(* IEC 61131-3 sources: OpenPLC_Sample_Programs/successed_ST (part 13) *)

(* ---- Scenario3v1_Final.st ---- *)
TYPE
    STATES_CRANE : (INIT, START_CRANE, CRANE_INIT, CRANE_INIT_2, INTERSTEP, INTERSTEP_2, TIMEDELAY, TURN_RIGHT, INTERSTEP_CHECK_WORKPIECE, CRANE_LOWER, STEP0, CRANE_LIFT_MAGAZIN, CRANE_TURN_LEFT_NOT_METALLIC, CRANE_ON_CONVEYOR, CRANE_LIFT_MAGAZIN_METALLIC, CRANE_TURN_LEFT_METALLIC, CRANE_ON_STAMP_METALLIC, RELEASE_WORKPIECE, CRANE_GO_UP, PAUSE, RESET_INTERCONNECT, LOWER_CRANE, SUCK_AT_STAMP, CRANE_LIFT_AT_STAMP, CRANE_TURN_LEFT_FROM_STAMP, CRANE_ON_CONVEYOR_METALLIC, RELEASE, CRANE_LIFT_CONVEYOR, WAIT_AT_STAMP, STEP2);
    STATES_MAGAZIN : (INIT, START_MAGAZIN, GREEN_LAMP, MAGAZIN_INIT, MAGAZIN_INIT_2, INTERSTEP, CONVEY, STEP0, SLIDER_MOVE_BACK, STEP1);
    STATES_STAMP : (INIT, START_STAMP, GREEN_LAMP, STAMP_INIT_1, STAMP_INIT_2, STAMP_INIT_3, STAMP_INIT_4, INTERSTEP, INTERSTEP_2, STEP0, STAMPSLIDERBACK, STAMPPROCESS, STEP1, STAMPSLIDERFORWARD, STEP2);
END_TYPE

PROGRAM MAIN
    VAR_OUTPUT
        ACTUATOR_ANALOGCRANEPRESSURE : INT := INT#0;
        ACTUATOR_CRANELOWER : BOOL := FALSE;
        ACTUATOR_CRANETURNCLOCKWISE : BOOL := FALSE;
        ACTUATOR_CRANETURNCOUNTERCLOCKWISE : BOOL := FALSE;
        ACTUATOR_MAGAZINGREENLAMP : BOOL := FALSE;
        ACTUATOR_MAGAZINSLIDER : BOOL := FALSE;
        ACTUATOR_MAGAZINVACUUMOFF : BOOL := FALSE;
        ACTUATOR_MAGAZINVACUUMON : BOOL := FALSE;
        ACTUATOR_MAGAZINWHITELAMP : BOOL := FALSE;
        ACTUATOR_SOMEACTUATOR : BOOL := FALSE;
        ACTUATOR_STAMPGREENLAMP : BOOL := FALSE;
        ACTUATOR_STAMPPUSHER : BOOL := FALSE;
        ACTUATOR_STAMPSLIDERMOVEDIN : BOOL := FALSE;
        ACTUATOR_STAMPSLIDERMOVEDOUT : BOOL := FALSE;
        ACTUATOR_STAMPWHITELAMP : BOOL := FALSE;
    END_VAR

    VAR
        CRANE_CRANEDOWN : BOOL := FALSE;
        CRANE_CRANELOWER : BOOL := FALSE;
        CRANE_CRANEONCONVEYOR : BOOL := FALSE;
        CRANE_CRANEONMAGAZIN : BOOL := FALSE;
        CRANE_CRANEPOSITIONSTAMP : BOOL := FALSE;
        CRANE_CRANESUCKED : BOOL := FALSE;
        CRANE_CRANETURNCLOCKWISE : BOOL := FALSE;
        CRANE_CRANETURNCOUNTERCLOCKWISE : BOOL := FALSE;
        CRANE_CRANEUP : BOOL := FALSE;
        CRANE_DURATION1 : UINT := UINT#0;
        CRANE_MAGAZINCAPACITIVESENSOR : BOOL := FALSE;
        CRANE_MAGAZINVACUUMOFF : BOOL := FALSE;
        CRANE_MAGAZINVACUUMON : BOOL := FALSE;
        CRANE_SFCINIT : BOOL := FALSE;
        CRANE_SFCRESET : BOOL := FALSE;
        CRANE_SLIDERMOVEDOUT : BOOL := FALSE;
        CRANE_SLIDERNOTMOVEDOUT : BOOL := FALSE;
        CRANE_STAMPLOWERED : BOOL := FALSE;
        CRANE_STAMPSLIDERFILLED : BOOL := FALSE;
        CRANE_STARTBUTTONMAGAZIN : BOOL := FALSE;
        CRANE_STARTCOMMANDCRANE : BOOL := FALSE;
        CRANE_STARTVAR : BOOL := FALSE;
        CRANE_TIMEDELAY_TIMER_ET : UINT := UINT#0;
        CRANE_TIMEDELAY_TIMER_IN : BOOL := FALSE;
        CRANE_TIMEDELAY_TIMER_PT : UINT := UINT#0;
        CRANE_TIMEDELAY_TIMER_Q : BOOL := FALSE;
        CRANE_TIMEDELAY_TIMER_DURATION : UINT := UINT#0;
        CRANE_TIMEDELAY_TIMER_INTERCONNECT : BOOL := FALSE;
        CRANE_TIMER1_ET : UINT := UINT#0;
        CRANE_TIMER1_IN : BOOL := FALSE;
        CRANE_TIMER1_PT : UINT := UINT#0;
        CRANE_TIMER1_Q : BOOL := FALSE;
        CRANE_WORKPIECEREADY : BOOL := FALSE;
        CRANE_2_TRANSIT : BOOL := FALSE;
        CRANE_2STATE : STATES_CRANE := STATES_CRANE#INIT;
        CRANE_ACTUALTIME1 : UINT := UINT#0;
        CRANE_INTERCONNECT : BOOL := FALSE;
        CRANE_INTERCONNECTCRANESTARTCOMMAND : BOOL := FALSE;
        MAG_CRANEDOWN : BOOL := FALSE;
        MAG_CRANELOWER : BOOL := FALSE;
        MAG_CRANEONCONVEYOR : BOOL := FALSE;
        MAG_CRANEONMAGAZIN : BOOL := FALSE;
        MAG_CRANESUCKED : BOOL := FALSE;
        MAG_CRANETURNCLOCKWISE : BOOL := FALSE;
        MAG_CRANETURNCOUNTERCLOCKWISE : BOOL := FALSE;
        MAG_CRANEUP : BOOL := FALSE;
        MAG_MAGAZINGREENLAMP : BOOL := FALSE;
        MAG_MAGAZINSLIDER : BOOL := FALSE;
        MAG_MAGAZINVACUUMOFF : BOOL := FALSE;
        MAG_MAGAZINVACUUMON : BOOL := FALSE;
        MAG_MAGAZINWHITELAMP : BOOL := FALSE;
        MAG_SFCINIT : BOOL := FALSE;
        MAG_SFCRESET : BOOL := FALSE;
        MAG_SLIDERMOVEDOUT : BOOL := FALSE;
        MAG_SLIDERNOTMOVEDOUT : BOOL := FALSE;
        MAG_STARTBUTTONMAGAZIN : BOOL := FALSE;
        MAG_STARTCOMMANDMAGAZIN : BOOL := FALSE;
        MAG_STARTVAR : BOOL := FALSE;
        MAG_WORKPIECEREADY : BOOL := FALSE;
        MAG_2_TRANSIT : BOOL := FALSE;
        MAG_2STATE : STATES_MAGAZIN := STATES_MAGAZIN#INIT;
        MAG_INTERCONNECTMAGAZINSTARTCOMMAND : BOOL := FALSE;
        STAMP_CRANEDOWN : BOOL := FALSE;
        STAMP_CRANEONCONVEYOR : BOOL := FALSE;
        STAMP_CRANEPOSITIONSTAMP : BOOL := FALSE;
        STAMP_CRANESUCKED : BOOL := FALSE;
        STAMP_CRANEUP : BOOL := FALSE;
        STAMP_DURATION : UINT := UINT#0;
        STAMP_SFCINIT : BOOL := FALSE;
        STAMP_SFCRESET : BOOL := FALSE;
        STAMP_STAMPGREENLAMP : BOOL := FALSE;
        STAMP_STAMPLOWERED : BOOL := FALSE;
        STAMP_STAMPPRESSURE : BOOL := FALSE;
        STAMP_STAMPPUSHER : BOOL := FALSE;
        STAMP_STAMPSLIDERFILLED : BOOL := FALSE;
        STAMP_STAMPSLIDERMOVEDIN : BOOL := FALSE;
        STAMP_STAMPSLIDERMOVEDOUT : BOOL := FALSE;
        STAMP_STAMPSLIDERSENSORMOVEDIN : BOOL := FALSE;
        STAMP_STAMPSLIDERSENSORMOVEDOUT : BOOL := FALSE;
        STAMP_STAMPSTARTBUTTON : BOOL := FALSE;
        STAMP_STAMPUP : BOOL := FALSE;
        STAMP_STAMPWHITELAMP : BOOL := FALSE;
        STAMP_STARTCOMMANDSTAMP : BOOL := FALSE;
        STAMP_STARTVAR : BOOL := FALSE;
        STAMP_TIMER_ET : UINT := UINT#0;
        STAMP_TIMER_IN : BOOL := FALSE;
        STAMP_TIMER_PT : UINT := UINT#0;
        STAMP_TIMER_Q : BOOL := FALSE;
        STAMP_2_TRANSIT : BOOL := FALSE;
        STAMP_2STATE : STATES_STAMP := STATES_STAMP#INIT;
        STAMP_INTERCONNECT : BOOL := FALSE;
        STAMP_INTERCONNECTSTAMPSTARTCOMMAND : BOOL := FALSE;
    END_VAR

    VAR
        CRANE_SFCPAUSE : BOOL := FALSE;
        MAG_SFCPAUSE : BOOL := FALSE;
        STAMP_SFCPAUSE : BOOL := FALSE;
    END_VAR

    VAR_INPUT
        SENSOR_CRANEDOWN : BOOL := FALSE;
        SENSOR_CRANEONCONVEYOR : BOOL := FALSE;
        SENSOR_CRANEONMAGAZIN : BOOL := FALSE;
        SENSOR_CRANEPOSITION : BOOL := FALSE;
        SENSOR_CRANEPOSITIONSTAMP : BOOL := FALSE;
        SENSOR_CRANESUCKED : BOOL := FALSE;
        SENSOR_CRANEUP : BOOL := FALSE;
        SENSOR_MAGAZINCAPACITIVESENSOR : BOOL := FALSE;
        SENSOR_MAGAZINEMERGENCYSTOP : BOOL := FALSE;
        SENSOR_MAGAZINOPTICALSENSOR : BOOL := FALSE;
        SENSOR_MAGAZINSWITCHMANUELLAUTOMATIC : BOOL := FALSE;
        SENSOR_SLIDERMOVEDOUT : BOOL := FALSE;
        SENSOR_SLIDERNOTMOVEDOUT : BOOL := FALSE;
        SENSOR_STAMPEMERGENCYSTOP : BOOL := FALSE;
        SENSOR_STAMPLOWERED : BOOL := FALSE;
        SENSOR_STAMPSLIDERFILLED : BOOL := FALSE;
        SENSOR_STAMPSLIDERSENSORMOVEDIN : BOOL := FALSE;
        SENSOR_STAMPSLIDERSENSORMOVEDOUT : BOOL := FALSE;
        SENSOR_STAMPSTARTBUTTON : BOOL := FALSE;
        SENSOR_STAMPSWITCHMANUELLAUTOMATIC : BOOL := FALSE;
        SENSOR_STAMPUP : BOOL := FALSE;
        SENSOR_STARTBUTTONMAGAZIN : BOOL := FALSE;
        SENSOR_WORKPIECEREADY : BOOL := FALSE;
    END_VAR

    MAG_SLIDERNOTMOVEDOUT := SENSOR_SLIDERNOTMOVEDOUT;
    MAG_SLIDERMOVEDOUT := SENSOR_SLIDERMOVEDOUT;
    MAG_CRANEONMAGAZIN := SENSOR_CRANEONMAGAZIN;
    MAG_CRANEDOWN := SENSOR_CRANEDOWN;
    MAG_CRANEUP := SENSOR_CRANEUP;
    MAG_CRANEONCONVEYOR := SENSOR_CRANEONCONVEYOR;
    MAG_WORKPIECEREADY := SENSOR_WORKPIECEREADY;
    MAG_STARTBUTTONMAGAZIN := SENSOR_STARTBUTTONMAGAZIN;
    ACTUATOR_MAGAZINSLIDER := MAG_MAGAZINSLIDER;
    ACTUATOR_MAGAZINGREENLAMP := MAG_MAGAZINGREENLAMP;
    CRANE_CRANEUP := SENSOR_CRANEUP;
    CRANE_CRANEONCONVEYOR := SENSOR_CRANEONCONVEYOR;
    CRANE_CRANEDOWN := SENSOR_CRANEDOWN;
    CRANE_CRANESUCKED := SENSOR_CRANESUCKED;
    CRANE_CRANEONMAGAZIN := SENSOR_CRANEONMAGAZIN;
    CRANE_MAGAZINCAPACITIVESENSOR := SENSOR_MAGAZINCAPACITIVESENSOR;
    CRANE_CRANEPOSITIONSTAMP := SENSOR_CRANEPOSITIONSTAMP;
    CRANE_SLIDERMOVEDOUT := SENSOR_SLIDERMOVEDOUT;
    CRANE_WORKPIECEREADY := SENSOR_WORKPIECEREADY;
    CRANE_STAMPSLIDERFILLED := SENSOR_STAMPSLIDERFILLED;
    CRANE_SLIDERMOVEDOUT := SENSOR_SLIDERMOVEDOUT;
    CRANE_STARTBUTTONMAGAZIN := SENSOR_STARTBUTTONMAGAZIN;
    ACTUATOR_CRANETURNCOUNTERCLOCKWISE := CRANE_CRANETURNCOUNTERCLOCKWISE;
    ACTUATOR_CRANETURNCLOCKWISE := CRANE_CRANETURNCLOCKWISE;
    ACTUATOR_CRANELOWER := CRANE_CRANELOWER;
    ACTUATOR_MAGAZINVACUUMOFF := CRANE_MAGAZINVACUUMOFF;
    ACTUATOR_MAGAZINVACUUMON := CRANE_MAGAZINVACUUMON;
    STAMP_STAMPSLIDERSENSORMOVEDOUT := SENSOR_STAMPSLIDERSENSORMOVEDOUT;
    STAMP_STAMPSLIDERSENSORMOVEDIN := SENSOR_STAMPSLIDERSENSORMOVEDIN;
    STAMP_STAMPSLIDERFILLED := SENSOR_STAMPSLIDERFILLED;
    STAMP_STAMPUP := SENSOR_STAMPUP;
    STAMP_STAMPLOWERED := SENSOR_STAMPLOWERED;
    STAMP_CRANEDOWN := SENSOR_CRANEDOWN;
    STAMP_CRANEUP := SENSOR_CRANEUP;
    STAMP_CRANESUCKED := SENSOR_CRANESUCKED;
    STAMP_CRANEPOSITIONSTAMP := SENSOR_CRANEPOSITIONSTAMP;
    STAMP_CRANEONCONVEYOR := SENSOR_CRANEONCONVEYOR;
    STAMP_STAMPSTARTBUTTON := SENSOR_STAMPSTARTBUTTON;
    ACTUATOR_STAMPSLIDERMOVEDOUT := STAMP_STAMPSLIDERMOVEDOUT;
    ACTUATOR_STAMPSLIDERMOVEDIN := STAMP_STAMPSLIDERMOVEDIN;
    ACTUATOR_STAMPWHITELAMP := STAMP_STAMPWHITELAMP;
    ACTUATOR_STAMPPUSHER := STAMP_STAMPPUSHER;
    ACTUATOR_STAMPGREENLAMP := STAMP_STAMPGREENLAMP;
    ACTUATOR_ANALOGCRANEPRESSURE := INT#6000;
    IF (SENSOR_STAMPEMERGENCYSTOP AND SENSOR_MAGAZINEMERGENCYSTOP) THEN
        (* ! REGION MAG[MAG_SFCINIT, MAG_INTERCONNECTMAGAZINSTARTCOMMAND](MAG_CRANEDOWN, MAG_CRANEONCONVEYOR, MAG_CRANEONMAGAZIN, MAG_CRANESUCKED, MAG_CRANEUP, MAG_SFCRESET, MAG_SLIDERMOVEDOUT, MAG_SLIDERNOTMOVEDOUT, MAG_STARTBUTTONMAGAZIN, MAG_STARTVAR, MAG_WORKPIECEREADY) => (MAG_CRANELOWER, MAG_CRANETURNCLOCKWISE, MAG_CRANETURNCOUNTERCLOCKWISE, MAG_MAGAZINGREENLAMP, MAG_MAGAZINSLIDER, MAG_MAGAZINVACUUMOFF, MAG_MAGAZINVACUUMON, MAG_MAGAZINWHITELAMP, MAG_STARTCOMMANDMAGAZIN)
 *)            IF (MAG_SFCINIT OR MAG_SFCRESET) THEN
                MAG_CRANEDOWN := FALSE;
                MAG_CRANELOWER := FALSE;
                MAG_CRANEONCONVEYOR := FALSE;
                MAG_CRANEONMAGAZIN := FALSE;
                MAG_CRANESUCKED := FALSE;
                MAG_CRANETURNCLOCKWISE := FALSE;
                MAG_CRANETURNCOUNTERCLOCKWISE := FALSE;
                MAG_CRANEUP := FALSE;
                MAG_MAGAZINGREENLAMP := FALSE;
                MAG_MAGAZINSLIDER := FALSE;
                MAG_MAGAZINVACUUMOFF := FALSE;
                MAG_MAGAZINVACUUMON := FALSE;
                MAG_MAGAZINWHITELAMP := FALSE;
                MAG_SFCINIT := FALSE;
                MAG_SFCRESET := FALSE;
                MAG_SLIDERMOVEDOUT := FALSE;
                MAG_SLIDERNOTMOVEDOUT := FALSE;
                MAG_STARTBUTTONMAGAZIN := FALSE;
                MAG_STARTCOMMANDMAGAZIN := FALSE;
                MAG_STARTVAR := FALSE;
                MAG_WORKPIECEREADY := FALSE;
                MAG_2_TRANSIT := FALSE;
                MAG_2STATE := STATES_MAGAZIN#INIT;
                MAG_INTERCONNECTMAGAZINSTARTCOMMAND := FALSE;
            END_IF;
            IF NOT (MAG_SFCINIT OR MAG_SFCPAUSE) THEN
                (* RUNNING PIPELINE STEP: EDU.KIT.ITI.FORMAL.AUTOMATION.ST.INTRODUCESTATEENUMVARIABLE
 *)
                (* END OF: EDU.KIT.ITI.FORMAL.AUTOMATION.ST.INTRODUCESTATEENUMVARIABLE
 *)
                (* RUNNING PIPELINE STEP: EDU.KIT.ITI.FORMAL.AUTOMATION.ST.TRANSLATIONSFCTOSTOLD_INTRODUCETRANSITVARIABLE
 *)
                (* END OF: EDU.KIT.ITI.FORMAL.AUTOMATION.ST.TRANSLATIONSFCTOSTOLD_INTRODUCETRANSITVARIABLE
 *)
                (* RUNNING PIPELINE STEP: EDU.KIT.ITI.FORMAL.AUTOMATION.ST.TRANSLATIONSFCTOSTOLD_THEBIGSTATECASE
 *)
                CASE MAG_2STATE OF
                    STATES_MAGAZIN#INIT:
                        MAG_2_TRANSIT := FALSE;
                        IF TRUE THEN
                            MAG_2_TRANSIT := TRUE;
                            MAG_2STATE := STATES_MAGAZIN#START_MAGAZIN;
                        END_IF;

                    STATES_MAGAZIN#START_MAGAZIN:
                        MAG_2_TRANSIT := FALSE;
                        (* CALL OF ACTION: START_MAGAZIN_ACTIVE
 *)
                        MAG_MAGAZINSLIDER := FALSE;
                        MAG_MAGAZINGREENLAMP := FALSE;
                        MAG_STARTVAR := FALSE;
                        MAG_STARTCOMMANDMAGAZIN := FALSE;
                        IF (MAG_STARTBUTTONMAGAZIN = TRUE) THEN
                            MAG_INTERCONNECTMAGAZINSTARTCOMMAND := TRUE;
                        END_IF;
                        (* END OF ACTION CALL: START_MAGAZIN_ACTIVE
 *)
                        IF MAG_INTERCONNECTMAGAZINSTARTCOMMAND THEN
                            MAG_2_TRANSIT := TRUE;
                            MAG_2STATE := STATES_MAGAZIN#GREEN_LAMP;
                        END_IF;

                    STATES_MAGAZIN#GREEN_LAMP:
                        MAG_2_TRANSIT := FALSE;
                        (* CALL OF ACTION: GREEN_LAMP_ACTIVE
 *)
                        MAG_MAGAZINGREENLAMP := TRUE;
                        MAG_INTERCONNECTMAGAZINSTARTCOMMAND := FALSE;
                        (* END OF ACTION CALL: GREEN_LAMP_ACTIVE
 *)
                        IF TRUE THEN
                            MAG_2_TRANSIT := TRUE;
                            MAG_2STATE := STATES_MAGAZIN#MAGAZIN_INIT;
                        END_IF;

                    STATES_MAGAZIN#MAGAZIN_INIT:
                        MAG_2_TRANSIT := FALSE;
                        (* CALL OF ACTION: MAGAZIN_INIT_ACTIVE
 *)
                        MAG_MAGAZINSLIDER := TRUE;
                        (* END OF ACTION CALL: MAGAZIN_INIT_ACTIVE
 *)
                        IF TRUE THEN
                            MAG_2_TRANSIT := TRUE;
                            MAG_2STATE := STATES_MAGAZIN#MAGAZIN_INIT_2;
                        END_IF;

                    STATES_MAGAZIN#MAGAZIN_INIT_2:
                        MAG_2_TRANSIT := FALSE;
                        (* CALL OF ACTION: MAGAZIN_INIT_2_ACTIVE
 *)
                        MAG_MAGAZINSLIDER := FALSE;
                        (* END OF ACTION CALL: MAGAZIN_INIT_2_ACTIVE
 *)
                        IF TRUE THEN
                            MAG_2_TRANSIT := TRUE;
                            MAG_2STATE := STATES_MAGAZIN#INTERSTEP;
                        END_IF;

                    STATES_MAGAZIN#INTERSTEP:
                        MAG_2_TRANSIT := FALSE;
                        (* CALL OF ACTION: INTERSTEP_ACTIVE
 *)
                        MAG_STARTCOMMANDMAGAZIN := TRUE;
                        (* END OF ACTION CALL: INTERSTEP_ACTIVE
 *)
                        IF MAG_STARTVAR THEN
                            MAG_2_TRANSIT := TRUE;
                            MAG_2STATE := STATES_MAGAZIN#CONVEY;
                        END_IF;

                    STATES_MAGAZIN#CONVEY:
                        MAG_2_TRANSIT := FALSE;
                        (* CALL OF ACTION: CONVEY_ACTIVE
 *)
                        IF MAG_SLIDERNOTMOVEDOUT THEN
                            MAG_MAGAZINSLIDER := TRUE;
                        END_IF;
                        (* END OF ACTION CALL: CONVEY_ACTIVE
 *)
                        IF MAG_CRANEONMAGAZIN THEN
                            MAG_2_TRANSIT := TRUE;
                            MAG_2STATE := STATES_MAGAZIN#STEP0;
                        END_IF;

                    STATES_MAGAZIN#STEP0:
                        MAG_2_TRANSIT := FALSE;
                        IF MAG_CRANEDOWN THEN
                            MAG_2_TRANSIT := TRUE;
                            MAG_2STATE := STATES_MAGAZIN#SLIDER_MOVE_BACK;
                        END_IF;

                    STATES_MAGAZIN#SLIDER_MOVE_BACK:
                        MAG_2_TRANSIT := FALSE;
                        (* CALL OF ACTION: SLIDERMOVEBACK_ACTIVE
 *)
                        IF ((MAG_SLIDERMOVEDOUT = TRUE) AND (MAG_SLIDERNOTMOVEDOUT = FALSE)) THEN
                            MAG_MAGAZINSLIDER := FALSE;
                        END_IF;
                        (* END OF ACTION CALL: SLIDERMOVEBACK_ACTIVE
 *)
                        IF MAG_CRANEUP THEN
                            MAG_2_TRANSIT := TRUE;
                            MAG_2STATE := STATES_MAGAZIN#STEP1;
                        END_IF;

                    STATES_MAGAZIN#STEP1:
                        MAG_2_TRANSIT := FALSE;
                        IF MAG_CRANEONCONVEYOR THEN
                            MAG_2_TRANSIT := TRUE;
                            MAG_2STATE := STATES_MAGAZIN#INTERSTEP;
                        END_IF;

                                    END_CASE;
                (* END OF: EDU.KIT.ITI.FORMAL.AUTOMATION.ST.TRANSLATIONSFCTOSTOLD_THEBIGSTATECASE
 *)
                (* RUNNING PIPELINE STEP: EDU.KIT.ITI.FORMAL.AUTOMATION.ST.SFCFLAGINTRODUCTION
 *)
            END_IF;
            (* END OF: EDU.KIT.ITI.FORMAL.AUTOMATION.ST.SFCFLAGINTRODUCTION
 *)
        (* ! END_REGION
 *)        (* ! REGION CRANE[CRANE_DURATION1, CRANE_SFCINIT, CRANE_TIMEDELAY_TIMER_ET, CRANE_TIMEDELAY_TIMER_IN, CRANE_TIMEDELAY_TIMER_PT, CRANE_TIMEDELAY_TIMER_Q, CRANE_TIMEDELAY_TIMER_DURATION, CRANE_TIMEDELAY_TIMER_INTERCONNECT, CRANE_TIMER1_ET, CRANE_TIMER1_IN, CRANE_TIMER1_PT, CRANE_TIMER1_Q, CRANE_ACTUALTIME1, CRANE_INTERCONNECT, CRANE_INTERCONNECTCRANESTARTCOMMAND](CRANE_CRANEDOWN, CRANE_CRANEONCONVEYOR, CRANE_CRANEONMAGAZIN, CRANE_CRANEPOSITIONSTAMP, CRANE_CRANESUCKED, CRANE_CRANEUP, CRANE_MAGAZINCAPACITIVESENSOR, CRANE_SFCRESET, CRANE_SLIDERMOVEDOUT, CRANE_SLIDERNOTMOVEDOUT, CRANE_STAMPLOWERED, CRANE_STAMPSLIDERFILLED, CRANE_STARTBUTTONMAGAZIN, CRANE_STARTVAR, CRANE_WORKPIECEREADY) => (CRANE_CRANELOWER, CRANE_CRANETURNCLOCKWISE, CRANE_CRANETURNCOUNTERCLOCKWISE, CRANE_MAGAZINVACUUMOFF, CRANE_MAGAZINVACUUMON, CRANE_STARTCOMMANDCRANE)
 *)            IF (CRANE_SFCINIT OR CRANE_SFCRESET) THEN
                CRANE_CRANEDOWN := FALSE;
                CRANE_CRANELOWER := FALSE;
                CRANE_CRANEONCONVEYOR := FALSE;
                CRANE_CRANEONMAGAZIN := FALSE;
                CRANE_CRANEPOSITIONSTAMP := FALSE;
                CRANE_CRANESUCKED := FALSE;
                CRANE_CRANETURNCLOCKWISE := FALSE;
                CRANE_CRANETURNCOUNTERCLOCKWISE := FALSE;
                CRANE_CRANEUP := FALSE;
                CRANE_DURATION1 := UINT#375;
                CRANE_MAGAZINCAPACITIVESENSOR := FALSE;
                CRANE_MAGAZINVACUUMOFF := FALSE;
                CRANE_MAGAZINVACUUMON := FALSE;
                CRANE_SFCINIT := FALSE;
                CRANE_SFCRESET := FALSE;
                CRANE_SLIDERMOVEDOUT := FALSE;
                CRANE_SLIDERNOTMOVEDOUT := FALSE;
                CRANE_STAMPLOWERED := FALSE;
                CRANE_STAMPSLIDERFILLED := FALSE;
                CRANE_STARTBUTTONMAGAZIN := FALSE;
                CRANE_STARTCOMMANDCRANE := FALSE;
                CRANE_STARTVAR := FALSE;
                CRANE_TIMEDELAY_TIMER_ET := UINT#0;
                CRANE_TIMEDELAY_TIMER_IN := FALSE;
                CRANE_TIMEDELAY_TIMER_PT := UINT#0;
                CRANE_TIMEDELAY_TIMER_Q := FALSE;
                CRANE_TIMEDELAY_TIMER_DURATION := UINT#12;
                CRANE_TIMEDELAY_TIMER_INTERCONNECT := FALSE;
                CRANE_TIMER1_ET := UINT#0;
                CRANE_TIMER1_IN := FALSE;
                CRANE_TIMER1_PT := UINT#0;
                CRANE_TIMER1_Q := FALSE;
                CRANE_WORKPIECEREADY := FALSE;
                CRANE_2_TRANSIT := FALSE;
                CRANE_2STATE := STATES_CRANE#INIT;
                CRANE_ACTUALTIME1 := UINT#0;
                CRANE_INTERCONNECT := FALSE;
                CRANE_INTERCONNECTCRANESTARTCOMMAND := FALSE;
            END_IF;
            IF NOT (CRANE_SFCINIT OR CRANE_SFCPAUSE) THEN
                (* RUNNING PIPELINE STEP: EDU.KIT.ITI.FORMAL.AUTOMATION.ST.INTRODUCESTATEENUMVARIABLE
 *)
                (* END OF: EDU.KIT.ITI.FORMAL.AUTOMATION.ST.INTRODUCESTATEENUMVARIABLE
 *)
                (* RUNNING PIPELINE STEP: EDU.KIT.ITI.FORMAL.AUTOMATION.ST.TRANSLATIONSFCTOSTOLD_INTRODUCETRANSITVARIABLE
 *)
                (* END OF: EDU.KIT.ITI.FORMAL.AUTOMATION.ST.TRANSLATIONSFCTOSTOLD_INTRODUCETRANSITVARIABLE
 *)
                (* RUNNING PIPELINE STEP: EDU.KIT.ITI.FORMAL.AUTOMATION.ST.TRANSLATIONSFCTOSTOLD_THEBIGSTATECASE
 *)
                CASE CRANE_2STATE OF
                    STATES_CRANE#INIT:
                        CRANE_2_TRANSIT := FALSE;
                        IF TRUE THEN
                            CRANE_2_TRANSIT := TRUE;
                            CRANE_2STATE := STATES_CRANE#START_CRANE;
                        END_IF;

                    STATES_CRANE#START_CRANE:
                        CRANE_2_TRANSIT := FALSE;
                        (* CALL OF ACTION: START_CRANE_ACTIVE
 *)
                        CRANE_CRANELOWER := FALSE;
                        CRANE_MAGAZINVACUUMOFF := TRUE;
                        CRANE_MAGAZINVACUUMON := FALSE;
                        CRANE_CRANETURNCOUNTERCLOCKWISE := FALSE;
                        CRANE_CRANETURNCLOCKWISE := FALSE;
                        CRANE_STARTVAR := FALSE;
                        CRANE_STARTCOMMANDCRANE := FALSE;
                        IF (CRANE_STARTBUTTONMAGAZIN = TRUE) THEN
                            CRANE_INTERCONNECTCRANESTARTCOMMAND := TRUE;
                        END_IF;
                        (* END OF ACTION CALL: START_CRANE_ACTIVE
 *)
                        IF CRANE_INTERCONNECTCRANESTARTCOMMAND THEN
                            CRANE_2_TRANSIT := TRUE;
                            CRANE_2STATE := STATES_CRANE#CRANE_INIT;
                        END_IF;

                    STATES_CRANE#CRANE_INIT:
                        CRANE_2_TRANSIT := FALSE;
                        (* CALL OF ACTION: CRANE_INIT_ACTIVE
 *)
                        CRANE_CRANELOWER := TRUE;
                        CRANE_INTERCONNECTCRANESTARTCOMMAND := FALSE;
                        (* END OF ACTION CALL: CRANE_INIT_ACTIVE
 *)
                        IF CRANE_CRANEDOWN THEN
                            CRANE_2_TRANSIT := TRUE;
                            CRANE_2STATE := STATES_CRANE#CRANE_INIT_2;
                        END_IF;

                    STATES_CRANE#CRANE_INIT_2:
                        CRANE_2_TRANSIT := FALSE;
                        (* CALL OF ACTION: CRANE_INIT_2_ACTIVE
 *)
                        CRANE_CRANELOWER := FALSE;
                        (* END OF ACTION CALL: CRANE_INIT_2_ACTIVE
 *)
                        IF CRANE_CRANEUP THEN
                            CRANE_2_TRANSIT := TRUE;
                            CRANE_2STATE := STATES_CRANE#INTERSTEP;
                        END_IF;

                    STATES_CRANE#INTERSTEP:
                        CRANE_2_TRANSIT := FALSE;
                        (* CALL OF ACTION: INTERSTEP_ACTIVE
 *)
                        CRANE_STARTCOMMANDCRANE := TRUE;
                        (* END OF ACTION CALL: INTERSTEP_ACTIVE
 *)
                        IF CRANE_STARTVAR THEN
                            CRANE_2_TRANSIT := TRUE;
                            CRANE_2STATE := STATES_CRANE#INTERSTEP_2;
                        END_IF;

                    STATES_CRANE#INTERSTEP_2:
                        CRANE_2_TRANSIT := FALSE;
                        IF CRANE_SLIDERMOVEDOUT THEN
                            CRANE_2_TRANSIT := TRUE;
                            CRANE_2STATE := STATES_CRANE#TIMEDELAY;
                        END_IF;

                    STATES_CRANE#TIMEDELAY:
                        CRANE_2_TRANSIT := FALSE;
                        (* CALL OF ACTION: TIMEDELAY_ACTIVE
 *)
                        CRANE_TIMEDELAY_TIMER_IN := TRUE;
                        CRANE_TIMEDELAY_TIMER_PT := CRANE_TIMEDELAY_TIMER_DURATION;
                        (* ! REGION TIMEDELAY_TIMER[](CRANE_TIMEDELAY_TIMER_IN, CRANE_TIMEDELAY_TIMER_PT) => (CRANE_TIMEDELAY_TIMER_ET, CRANE_TIMEDELAY_TIMER_Q)
 *)                            IF CRANE_TIMEDELAY_TIMER_IN THEN
                                CRANE_TIMEDELAY_TIMER_Q := (CRANE_TIMEDELAY_TIMER_ET = UINT#0);
                                IF (CRANE_TIMEDELAY_TIMER_ET > UINT#0) THEN
                                    CRANE_TIMEDELAY_TIMER_ET := (CRANE_TIMEDELAY_TIMER_ET - UINT#1);
                                ELSE
                                    CRANE_TIMEDELAY_TIMER_ET := UINT#0;
                                END_IF;
                            ELSE
                                CRANE_TIMEDELAY_TIMER_Q := FALSE;
                                CRANE_TIMEDELAY_TIMER_ET := CRANE_TIMEDELAY_TIMER_PT;
                            END_IF;
                        (* ! END_REGION
 *)                        CRANE_TIMEDELAY_TIMER_INTERCONNECT := CRANE_TIMEDELAY_TIMER_Q;
                        (* END OF ACTION CALL: TIMEDELAY_ACTIVE
 *)
                        IF CRANE_TIMEDELAY_TIMER_INTERCONNECT THEN
                            CRANE_2_TRANSIT := TRUE;
                            CRANE_2STATE := STATES_CRANE#TURN_RIGHT;
                        END_IF;

                    STATES_CRANE#TURN_RIGHT:
                        CRANE_2_TRANSIT := FALSE;
                        (* CALL OF ACTION: STEP0_ACTIVE
 *)
                        CRANE_CRANETURNCLOCKWISE := TRUE;
                        CRANE_CRANETURNCOUNTERCLOCKWISE := FALSE;
                        (* END OF ACTION CALL: STEP0_ACTIVE
 *)
                        IF CRANE_CRANEONMAGAZIN THEN
                            CRANE_2_TRANSIT := TRUE;
                            CRANE_2STATE := STATES_CRANE#INTERSTEP_CHECK_WORKPIECE;
                        END_IF;

                    STATES_CRANE#INTERSTEP_CHECK_WORKPIECE:
                        CRANE_2_TRANSIT := FALSE;
                        (* CALL OF ACTION: INTERSTEP_CHECK_WORKPIECE_ACTIVE
 *)
                        CRANE_CRANETURNCLOCKWISE := FALSE;
                        CRANE_CRANETURNCOUNTERCLOCKWISE := FALSE;
                        (* END OF ACTION CALL: INTERSTEP_CHECK_WORKPIECE_ACTIVE
 *)
                        IF CRANE_WORKPIECEREADY THEN
                            CRANE_2_TRANSIT := TRUE;
                            CRANE_2STATE := STATES_CRANE#CRANE_LOWER;
                        ELSIF (NOT CRANE_WORKPIECEREADY AND CRANE_STAMPSLIDERFILLED) THEN
                            CRANE_2_TRANSIT := TRUE;
                            CRANE_2STATE := STATES_CRANE#WAIT_AT_STAMP;
                        ELSIF (NOT CRANE_WORKPIECEREADY AND NOT CRANE_STAMPSLIDERFILLED) THEN
                            CRANE_2_TRANSIT := TRUE;
                            CRANE_2STATE := STATES_CRANE#STEP2;
                        END_IF;

                    STATES_CRANE#CRANE_LOWER:
                        CRANE_2_TRANSIT := FALSE;
                        (* CALL OF ACTION: MAGAZINSTOP_ACTIVE
 *)
                        CRANE_MAGAZINVACUUMON := TRUE;
                        CRANE_MAGAZINVACUUMOFF := FALSE;
                        CRANE_CRANELOWER := TRUE;
                        (* END OF ACTION CALL: MAGAZINSTOP_ACTIVE
 *)
                        IF CRANE_CRANESUCKED THEN
                            CRANE_2_TRANSIT := TRUE;
                            CRANE_2STATE := STATES_CRANE#STEP0;
                        END_IF;

                    STATES_CRANE#STEP0:
                        CRANE_2_TRANSIT := FALSE;
                        IF NOT CRANE_MAGAZINCAPACITIVESENSOR THEN
                            CRANE_2_TRANSIT := TRUE;
                            CRANE_2STATE := STATES_CRANE#CRANE_LIFT_MAGAZIN;
                        ELSIF CRANE_MAGAZINCAPACITIVESENSOR THEN
                            CRANE_2_TRANSIT := TRUE;
                            CRANE_2STATE := STATES_CRANE#CRANE_LIFT_MAGAZIN_METALLIC;
                        END_IF;

                    STATES_CRANE#CRANE_LIFT_MAGAZIN:
                        CRANE_2_TRANSIT := FALSE;
                        (* CALL OF ACTION: CRANELIFTMAGAZIN_ACTIVE
 *)
                        CRANE_CRANELOWER := FALSE;
                        (* END OF ACTION CALL: CRANELIFTMAGAZIN_ACTIVE
 *)
                        IF CRANE_CRANEUP THEN
                            CRANE_2_TRANSIT := TRUE;
                            CRANE_2STATE := STATES_CRANE#CRANE_TURN_LEFT_NOT_METALLIC;
                        END_IF;

                    STATES_CRANE#CRANE_TURN_LEFT_NOT_METALLIC:
                        CRANE_2_TRANSIT := FALSE;
                        (* CALL OF ACTION: CRANETURNLEFT_ACTIVE
 *)
                        CRANE_CRANETURNCOUNTERCLOCKWISE := TRUE;
                        CRANE_CRANETURNCLOCKWISE := FALSE;
                        (* END OF ACTION CALL: CRANETURNLEFT_ACTIVE
 *)
                        IF CRANE_CRANEONCONVEYOR THEN
                            CRANE_2_TRANSIT := TRUE;
                            CRANE_2STATE := STATES_CRANE#CRANE_ON_CONVEYOR;
                        END_IF;

                    STATES_CRANE#CRANE_ON_CONVEYOR:
                        CRANE_2_TRANSIT := FALSE;
                        (* CALL OF ACTION: CRANEONCONVEYOR_ACTIVE
 *)
                        CRANE_CRANETURNCOUNTERCLOCKWISE := FALSE;
                        CRANE_CRANETURNCLOCKWISE := FALSE;
                        CRANE_CRANELOWER := TRUE;
                        (* END OF ACTION CALL: CRANEONCONVEYOR_ACTIVE
 *)
                        IF CRANE_CRANEDOWN THEN
                            CRANE_2_TRANSIT := TRUE;
                            CRANE_2STATE := STATES_CRANE#RELEASE;
                        END_IF;

                    STATES_CRANE#CRANE_LIFT_MAGAZIN_METALLIC:
                        CRANE_2_TRANSIT := FALSE;
                        (* CALL OF ACTION: CRANE_LIFT_MAGAZIN_METALLIC_ACTIVE_0
 *)
                        CRANE_CRANELOWER := FALSE;
                        (* END OF ACTION CALL: CRANE_LIFT_MAGAZIN_METALLIC_ACTIVE_0
 *)
                        IF CRANE_CRANEUP THEN
                            CRANE_2_TRANSIT := TRUE;
                            CRANE_2STATE := STATES_CRANE#CRANE_TURN_LEFT_METALLIC;
                        END_IF;

                    STATES_CRANE#CRANE_TURN_LEFT_METALLIC:
                        CRANE_2_TRANSIT := FALSE;
                        (* CALL OF ACTION: CRANE_TURN_LEFT_METALLIC_ACTIVE
 *)
                        CRANE_CRANETURNCOUNTERCLOCKWISE := TRUE;
                        CRANE_CRANETURNCLOCKWISE := FALSE;
                        (* END OF ACTION CALL: CRANE_TURN_LEFT_METALLIC_ACTIVE
 *)
                        IF CRANE_CRANEPOSITIONSTAMP THEN
                            CRANE_2_TRANSIT := TRUE;
                            CRANE_2STATE := STATES_CRANE#CRANE_ON_STAMP_METALLIC;
                        END_IF;

                    STATES_CRANE#CRANE_ON_STAMP_METALLIC:
                        CRANE_2_TRANSIT := FALSE;
                        (* CALL OF ACTION: CRANE_ON_CONVEYOR_METALLIC_ACTIVE
 *)
                        CRANE_CRANETURNCOUNTERCLOCKWISE := FALSE;
                        CRANE_CRANETURNCLOCKWISE := FALSE;
                        CRANE_CRANELOWER := TRUE;
                        (* END OF ACTION CALL: CRANE_ON_CONVEYOR_METALLIC_ACTIVE
 *)
                        IF CRANE_CRANEDOWN THEN
                            CRANE_2_TRANSIT := TRUE;
                            CRANE_2STATE := STATES_CRANE#RELEASE_WORKPIECE;
                        END_IF;

                    STATES_CRANE#RELEASE_WORKPIECE:
                        CRANE_2_TRANSIT := FALSE;
                        (* CALL OF ACTION: RELEASE_WORKPIECE_ACTIVE
 *)
                        CRANE_MAGAZINVACUUMOFF := TRUE;
                        CRANE_MAGAZINVACUUMON := FALSE;
                        (* END OF ACTION CALL: RELEASE_WORKPIECE_ACTIVE
 *)
                        IF TRUE THEN
                            CRANE_2_TRANSIT := TRUE;
                            CRANE_2STATE := STATES_CRANE#CRANE_GO_UP;
                        END_IF;

                    STATES_CRANE#CRANE_GO_UP:
                        CRANE_2_TRANSIT := FALSE;
                        (* CALL OF ACTION: CRANE_GO_UP_ACTIVE
 *)
                        CRANE_CRANELOWER := FALSE;
                        (* END OF ACTION CALL: CRANE_GO_UP_ACTIVE
 *)
                        IF CRANE_CRANEUP THEN
                            CRANE_2_TRANSIT := TRUE;
                            CRANE_2STATE := STATES_CRANE#PAUSE;
                        END_IF;

                    STATES_CRANE#PAUSE:
                        CRANE_2_TRANSIT := FALSE;
                        (* CALL OF ACTION: PAUSE_ACTIVE
 *)
                        CRANE_TIMER1_IN := CRANE_CRANEUP;
                        CRANE_TIMER1_PT := CRANE_DURATION1;
                        (* ! REGION TIMER1[](CRANE_TIMER1_IN, CRANE_TIMER1_PT) => (CRANE_TIMER1_ET, CRANE_TIMER1_Q)
 *)                            IF CRANE_TIMER1_IN THEN
                                CRANE_TIMER1_Q := (CRANE_TIMER1_ET = UINT#0);
                                IF (CRANE_TIMER1_ET > UINT#0) THEN
                                    CRANE_TIMER1_ET := (CRANE_TIMER1_ET - UINT#1);
                                ELSE
                                    CRANE_TIMER1_ET := UINT#0;
                                END_IF;
                            ELSE
                                CRANE_TIMER1_Q := FALSE;
                                CRANE_TIMER1_ET := CRANE_TIMER1_PT;
                            END_IF;
                        (* ! END_REGION
 *)                        CRANE_INTERCONNECT := CRANE_TIMER1_Q;
                        (* END OF ACTION CALL: PAUSE_ACTIVE
 *)
                        IF CRANE_INTERCONNECT THEN
                            CRANE_2_TRANSIT := TRUE;
                            CRANE_2STATE := STATES_CRANE#RESET_INTERCONNECT;
                        END_IF;

                    STATES_CRANE#RESET_INTERCONNECT:
                        CRANE_2_TRANSIT := FALSE;
                        (* CALL OF ACTION: RESET_INTERCONNECT_ACTIVE
 *)
                        CRANE_INTERCONNECT := FALSE;
                        CRANE_TIMER1_IN := FALSE;
                        CRANE_TIMER1_PT := UINT#0;
                        (* ! REGION TIMER1[](CRANE_TIMER1_IN, CRANE_TIMER1_PT) => (CRANE_TIMER1_ET, CRANE_TIMER1_Q)
 *)                            IF CRANE_TIMER1_IN THEN
                                CRANE_TIMER1_Q := (CRANE_TIMER1_ET = UINT#0);
                                IF (CRANE_TIMER1_ET > UINT#0) THEN
                                    CRANE_TIMER1_ET := (CRANE_TIMER1_ET - UINT#1);
                                ELSE
                                    CRANE_TIMER1_ET := UINT#0;
                                END_IF;
                            ELSE
                                CRANE_TIMER1_Q := FALSE;
                                CRANE_TIMER1_ET := CRANE_TIMER1_PT;
                            END_IF;
                        (* ! END_REGION
 *)                        (* END OF ACTION CALL: RESET_INTERCONNECT_ACTIVE
 *)
                        IF CRANE_SLIDERMOVEDOUT THEN
                            CRANE_2_TRANSIT := TRUE;
                            CRANE_2STATE := STATES_CRANE#LOWER_CRANE;
                        END_IF;

                    STATES_CRANE#LOWER_CRANE:
                        CRANE_2_TRANSIT := FALSE;
                        (* CALL OF ACTION: LOWER_CRANE_ACTIVE
 *)
                        CRANE_CRANELOWER := TRUE;
                        (* END OF ACTION CALL: LOWER_CRANE_ACTIVE
 *)
                        IF CRANE_CRANEDOWN THEN
                            CRANE_2_TRANSIT := TRUE;
                            CRANE_2STATE := STATES_CRANE#SUCK_AT_STAMP;
                        END_IF;

                    STATES_CRANE#SUCK_AT_STAMP:
                        CRANE_2_TRANSIT := FALSE;
                        (* CALL OF ACTION: SUCK_AT_STAMP_ACTIVE
 *)
                        CRANE_MAGAZINVACUUMON := TRUE;
                        CRANE_MAGAZINVACUUMOFF := FALSE;
                        (* END OF ACTION CALL: SUCK_AT_STAMP_ACTIVE
 *)
                        IF CRANE_CRANESUCKED THEN
                            CRANE_2_TRANSIT := TRUE;
                            CRANE_2STATE := STATES_CRANE#CRANE_LIFT_AT_STAMP;
                        END_IF;

                    STATES_CRANE#CRANE_LIFT_AT_STAMP:
                        CRANE_2_TRANSIT := FALSE;
                        (* CALL OF ACTION: CRANE_LIFT_AT_STAMP_ACTIVE
 *)
                        CRANE_CRANELOWER := FALSE;
                        (* END OF ACTION CALL: CRANE_LIFT_AT_STAMP_ACTIVE
 *)
                        IF CRANE_CRANEUP THEN
                            CRANE_2_TRANSIT := TRUE;
                            CRANE_2STATE := STATES_CRANE#CRANE_TURN_LEFT_FROM_STAMP;
                        END_IF;

                    STATES_CRANE#CRANE_TURN_LEFT_FROM_STAMP:
                        CRANE_2_TRANSIT := FALSE;
                        (* CALL OF ACTION: CRANE_TURN_LEFT_FROM_STAMP_ACTIVE
 *)
                        CRANE_CRANETURNCLOCKWISE := TRUE;
                        CRANE_CRANETURNCOUNTERCLOCKWISE := FALSE;
                        (* END OF ACTION CALL: CRANE_TURN_LEFT_FROM_STAMP_ACTIVE
 *)
                        IF CRANE_CRANEONCONVEYOR THEN
                            CRANE_2_TRANSIT := TRUE;
                            CRANE_2STATE := STATES_CRANE#CRANE_ON_CONVEYOR_METALLIC;
                        END_IF;

                    STATES_CRANE#CRANE_ON_CONVEYOR_METALLIC:
                        CRANE_2_TRANSIT := FALSE;
                        (* CALL OF ACTION: CRANE_ON_CONVEYOR_METALLIC_ACTIVE_0
 *)
                        CRANE_CRANETURNCOUNTERCLOCKWISE := FALSE;
                        CRANE_CRANETURNCLOCKWISE := FALSE;
                        CRANE_CRANELOWER := TRUE;
                        (* END OF ACTION CALL: CRANE_ON_CONVEYOR_METALLIC_ACTIVE_0
 *)
                        IF CRANE_CRANEDOWN THEN
                            CRANE_2_TRANSIT := TRUE;
                            CRANE_2STATE := STATES_CRANE#RELEASE;
                        END_IF;

                    STATES_CRANE#RELEASE:
                        CRANE_2_TRANSIT := FALSE;
                        (* CALL OF ACTION: RELEASE_ACTIVE
 *)
                        CRANE_MAGAZINVACUUMOFF := TRUE;
                        CRANE_MAGAZINVACUUMON := FALSE;
                        (* END OF ACTION CALL: RELEASE_ACTIVE
 *)
                        IF TRUE THEN
                            CRANE_2_TRANSIT := TRUE;
                            CRANE_2STATE := STATES_CRANE#CRANE_LIFT_CONVEYOR;
                        END_IF;

                    STATES_CRANE#CRANE_LIFT_CONVEYOR:
                        CRANE_2_TRANSIT := FALSE;
                        (* CALL OF ACTION: CRANELIFTCONVEYOR_ACTIVE
 *)
                        CRANE_CRANELOWER := FALSE;
                        (* END OF ACTION CALL: CRANELIFTCONVEYOR_ACTIVE
 *)
                        IF TRUE THEN
                            CRANE_2_TRANSIT := TRUE;
                            CRANE_2STATE := STATES_CRANE#INTERSTEP;
                        END_IF;

                    STATES_CRANE#WAIT_AT_STAMP:
                        CRANE_2_TRANSIT := FALSE;
                        IF TRUE THEN
                            CRANE_2_TRANSIT := TRUE;
                            CRANE_2STATE := STATES_CRANE#PAUSE;
                        END_IF;

                    STATES_CRANE#STEP2:
                        CRANE_2_TRANSIT := FALSE;
                        IF TRUE THEN
                            CRANE_2_TRANSIT := TRUE;
                            CRANE_2STATE := STATES_CRANE#START_CRANE;
                        END_IF;

                                    END_CASE;
                (* END OF: EDU.KIT.ITI.FORMAL.AUTOMATION.ST.TRANSLATIONSFCTOSTOLD_THEBIGSTATECASE
 *)
                (* RUNNING PIPELINE STEP: EDU.KIT.ITI.FORMAL.AUTOMATION.ST.SFCFLAGINTRODUCTION
 *)
            END_IF;
            (* END OF: EDU.KIT.ITI.FORMAL.AUTOMATION.ST.SFCFLAGINTRODUCTION
 *)
        (* ! END_REGION
 *)        (* ! REGION STAMP[STAMP_DURATION, STAMP_SFCINIT, STAMP_TIMER_ET, STAMP_TIMER_IN, STAMP_TIMER_PT, STAMP_TIMER_Q, STAMP_INTERCONNECT, STAMP_INTERCONNECTSTAMPSTARTCOMMAND](STAMP_CRANEDOWN, STAMP_CRANEONCONVEYOR, STAMP_CRANEPOSITIONSTAMP, STAMP_CRANESUCKED, STAMP_CRANEUP, STAMP_SFCRESET, STAMP_STAMPLOWERED, STAMP_STAMPSLIDERFILLED, STAMP_STAMPSLIDERSENSORMOVEDIN, STAMP_STAMPSLIDERSENSORMOVEDOUT, STAMP_STAMPSTARTBUTTON, STAMP_STAMPUP, STAMP_STARTVAR) => (STAMP_STAMPGREENLAMP, STAMP_STAMPPRESSURE, STAMP_STAMPPUSHER, STAMP_STAMPSLIDERMOVEDIN, STAMP_STAMPSLIDERMOVEDOUT, STAMP_STAMPWHITELAMP, STAMP_STARTCOMMANDSTAMP)
 *)            IF (STAMP_SFCINIT OR STAMP_SFCRESET) THEN
                STAMP_CRANEDOWN := FALSE;
                STAMP_CRANEONCONVEYOR := FALSE;
                STAMP_CRANEPOSITIONSTAMP := FALSE;
                STAMP_CRANESUCKED := FALSE;
                STAMP_CRANEUP := FALSE;
                STAMP_DURATION := UINT#125;
                STAMP_SFCINIT := FALSE;
                STAMP_SFCRESET := FALSE;
                STAMP_STAMPGREENLAMP := FALSE;
                STAMP_STAMPLOWERED := FALSE;
                STAMP_STAMPPRESSURE := FALSE;
                STAMP_STAMPPUSHER := FALSE;
                STAMP_STAMPSLIDERFILLED := FALSE;
                STAMP_STAMPSLIDERMOVEDIN := FALSE;
                STAMP_STAMPSLIDERMOVEDOUT := FALSE;
                STAMP_STAMPSLIDERSENSORMOVEDIN := FALSE;
                STAMP_STAMPSLIDERSENSORMOVEDOUT := FALSE;
                STAMP_STAMPSTARTBUTTON := FALSE;
                STAMP_STAMPUP := FALSE;
                STAMP_STAMPWHITELAMP := FALSE;
                STAMP_STARTCOMMANDSTAMP := FALSE;
                STAMP_STARTVAR := FALSE;
                STAMP_TIMER_ET := UINT#0;
                STAMP_TIMER_IN := FALSE;
                STAMP_TIMER_PT := UINT#0;
                STAMP_TIMER_Q := FALSE;
                STAMP_2_TRANSIT := FALSE;
                STAMP_2STATE := STATES_STAMP#INIT;
                STAMP_INTERCONNECT := FALSE;
                STAMP_INTERCONNECTSTAMPSTARTCOMMAND := FALSE;
            END_IF;
            IF NOT (STAMP_SFCINIT OR STAMP_SFCPAUSE) THEN
                (* RUNNING PIPELINE STEP: EDU.KIT.ITI.FORMAL.AUTOMATION.ST.INTRODUCESTATEENUMVARIABLE
 *)
                (* END OF: EDU.KIT.ITI.FORMAL.AUTOMATION.ST.INTRODUCESTATEENUMVARIABLE
 *)
                (* RUNNING PIPELINE STEP: EDU.KIT.ITI.FORMAL.AUTOMATION.ST.TRANSLATIONSFCTOSTOLD_INTRODUCETRANSITVARIABLE
 *)
                (* END OF: EDU.KIT.ITI.FORMAL.AUTOMATION.ST.TRANSLATIONSFCTOSTOLD_INTRODUCETRANSITVARIABLE
 *)
                (* RUNNING PIPELINE STEP: EDU.KIT.ITI.FORMAL.AUTOMATION.ST.TRANSLATIONSFCTOSTOLD_THEBIGSTATECASE
 *)
                CASE STAMP_2STATE OF
                    STATES_STAMP#INIT:
                        STAMP_2_TRANSIT := FALSE;
                        IF TRUE THEN
                            STAMP_2_TRANSIT := TRUE;
                            STAMP_2STATE := STATES_STAMP#START_STAMP;
                        END_IF;

                    STATES_STAMP#START_STAMP:
                        STAMP_2_TRANSIT := FALSE;
                        (* CALL OF ACTION: START_STAMP_ACTIVE
 *)
                        STAMP_STAMPSLIDERMOVEDOUT := FALSE;
                        STAMP_STAMPSLIDERMOVEDIN := FALSE;
                        STAMP_STAMPPUSHER := FALSE;
                        STAMP_STAMPGREENLAMP := FALSE;
                        STAMP_STAMPPRESSURE := FALSE;
                        STAMP_STARTCOMMANDSTAMP := FALSE;
                        IF (STAMP_STAMPSTARTBUTTON = TRUE) THEN
                            STAMP_INTERCONNECTSTAMPSTARTCOMMAND := TRUE;
                        END_IF;
                        (* END OF ACTION CALL: START_STAMP_ACTIVE
 *)
                        IF STAMP_INTERCONNECTSTAMPSTARTCOMMAND THEN
                            STAMP_2_TRANSIT := TRUE;
                            STAMP_2STATE := STATES_STAMP#GREEN_LAMP;
                        END_IF;

                    STATES_STAMP#GREEN_LAMP:
                        STAMP_2_TRANSIT := FALSE;
                        (* CALL OF ACTION: GREEN_LAMP_ACTIVE
 *)
                        STAMP_STAMPGREENLAMP := TRUE;
                        STAMP_INTERCONNECTSTAMPSTARTCOMMAND := FALSE;
                        (* END OF ACTION CALL: GREEN_LAMP_ACTIVE
 *)
                        IF TRUE THEN
                            STAMP_2_TRANSIT := TRUE;
                            STAMP_2STATE := STATES_STAMP#STAMP_INIT_1;
                        END_IF;

                    STATES_STAMP#STAMP_INIT_1:
                        STAMP_2_TRANSIT := FALSE;
                        (* CALL OF ACTION: STAMP_INIT_1_ACTIVE
 *)
                        STAMP_STAMPSLIDERMOVEDIN := TRUE;
                        STAMP_STAMPSLIDERMOVEDOUT := FALSE;
                        (* END OF ACTION CALL: STAMP_INIT_1_ACTIVE
 *)
                        IF STAMP_STAMPSLIDERSENSORMOVEDIN THEN
                            STAMP_2_TRANSIT := TRUE;
                            STAMP_2STATE := STATES_STAMP#STAMP_INIT_2;
                        END_IF;

                    STATES_STAMP#STAMP_INIT_2:
                        STAMP_2_TRANSIT := FALSE;
                        (* CALL OF ACTION: STAMP_INIT_2_ACTIVE
 *)
                        STAMP_STAMPSLIDERMOVEDIN := FALSE;
                        STAMP_STAMPSLIDERMOVEDOUT := TRUE;
                        (* END OF ACTION CALL: STAMP_INIT_2_ACTIVE
 *)
                        IF STAMP_STAMPSLIDERSENSORMOVEDOUT THEN
                            STAMP_2_TRANSIT := TRUE;
                            STAMP_2STATE := STATES_STAMP#STAMP_INIT_3;
                        END_IF;

                    STATES_STAMP#STAMP_INIT_3:
                        STAMP_2_TRANSIT := FALSE;
                        (* CALL OF ACTION: STAMP_INIT_3_ACTIVE
 *)
                        STAMP_STAMPPUSHER := TRUE;
                        (* END OF ACTION CALL: STAMP_INIT_3_ACTIVE
 *)
                        IF STAMP_STAMPLOWERED THEN
                            STAMP_2_TRANSIT := TRUE;
                            STAMP_2STATE := STATES_STAMP#STAMP_INIT_4;
                        END_IF;

                    STATES_STAMP#STAMP_INIT_4:
                        STAMP_2_TRANSIT := FALSE;
                        (* CALL OF ACTION: STAMP_INIT_4_ACTIVE
 *)
                        STAMP_STAMPPUSHER := FALSE;
                        (* END OF ACTION CALL: STAMP_INIT_4_ACTIVE
 *)
                        IF STAMP_STAMPUP THEN
                            STAMP_2_TRANSIT := TRUE;
                            STAMP_2STATE := STATES_STAMP#INTERSTEP;
                        END_IF;

                    STATES_STAMP#INTERSTEP:
                        STAMP_2_TRANSIT := FALSE;
                        (* CALL OF ACTION: INTERSTEP_ACTIVE
 *)
                        STAMP_STARTCOMMANDSTAMP := TRUE;
                        (* END OF ACTION CALL: INTERSTEP_ACTIVE
 *)
                        IF STAMP_STARTVAR THEN
                            STAMP_2_TRANSIT := TRUE;
                            STAMP_2STATE := STATES_STAMP#INTERSTEP_2;
                        END_IF;

                    STATES_STAMP#INTERSTEP_2:
                        STAMP_2_TRANSIT := FALSE;
                        IF STAMP_STAMPSLIDERFILLED THEN
                            STAMP_2_TRANSIT := TRUE;
                            STAMP_2STATE := STATES_STAMP#STEP0;
                        END_IF;

                    STATES_STAMP#STEP0:
                        STAMP_2_TRANSIT := FALSE;
                        IF STAMP_CRANEUP THEN
                            STAMP_2_TRANSIT := TRUE;
                            STAMP_2STATE := STATES_STAMP#STAMPSLIDERBACK;
                        END_IF;

                    STATES_STAMP#STAMPSLIDERBACK:
                        STAMP_2_TRANSIT := FALSE;
                        (* CALL OF ACTION: STAMPSLIDERBACK_ACTIVE
 *)
                        STAMP_STAMPSLIDERMOVEDIN := TRUE;
                        STAMP_STAMPSLIDERMOVEDOUT := FALSE;
                        (* END OF ACTION CALL: STAMPSLIDERBACK_ACTIVE
 *)
                        IF STAMP_STAMPSLIDERSENSORMOVEDIN THEN
                            STAMP_2_TRANSIT := TRUE;
                            STAMP_2STATE := STATES_STAMP#STAMPPROCESS;
                        END_IF;

                    STATES_STAMP#STAMPPROCESS:
                        STAMP_2_TRANSIT := FALSE;
                        (* CALL OF ACTION: STAMPPROCESS_ACTIVE
 *)
                        STAMP_STAMPSLIDERMOVEDIN := FALSE;
                        STAMP_STAMPPUSHER := TRUE;
                        (* END OF ACTION CALL: STAMPPROCESS_ACTIVE
 *)
                        IF STAMP_STAMPLOWERED THEN
                            STAMP_2_TRANSIT := TRUE;
                            STAMP_2STATE := STATES_STAMP#STEP1;
                        END_IF;

                    STATES_STAMP#STEP1:
                        STAMP_2_TRANSIT := FALSE;
                        (* CALL OF ACTION: STEP1_ACTIVE
 *)
                        STAMP_TIMER_IN := STAMP_STAMPLOWERED;
                        STAMP_TIMER_PT := UINT#0;
                        (* ! REGION TIMER[](STAMP_TIMER_IN, STAMP_TIMER_PT) => (STAMP_TIMER_ET, STAMP_TIMER_Q)
 *)                            IF STAMP_TIMER_IN THEN
                                STAMP_TIMER_Q := (STAMP_TIMER_ET = UINT#0);
                                IF (STAMP_TIMER_ET > UINT#0) THEN
                                    STAMP_TIMER_ET := (STAMP_TIMER_ET - UINT#1);
                                ELSE
                                    STAMP_TIMER_ET := UINT#0;
                                END_IF;
                            ELSE
                                STAMP_TIMER_Q := FALSE;
                                STAMP_TIMER_ET := STAMP_TIMER_PT;
                            END_IF;
                        (* ! END_REGION
 *)                        STAMP_INTERCONNECT := STAMP_TIMER_Q;
                        (* END OF ACTION CALL: STEP1_ACTIVE
 *)
                        IF STAMP_INTERCONNECT THEN
                            STAMP_2_TRANSIT := TRUE;
                            STAMP_2STATE := STATES_STAMP#STAMPSLIDERFORWARD;
                        END_IF;

                    STATES_STAMP#STAMPSLIDERFORWARD:
                        STAMP_2_TRANSIT := FALSE;
                        (* CALL OF ACTION: STAMPSLIDERFORWARD_ACTIVE
 *)
                        STAMP_STAMPPUSHER := FALSE;
                        STAMP_STAMPSLIDERMOVEDOUT := TRUE;
                        IF ((STAMP_STAMPLOWERED = FALSE) AND (STAMP_STAMPUP = TRUE)) THEN
                            STAMP_INTERCONNECT := FALSE;
                        END_IF;
                        STAMP_TIMER_IN := FALSE;
                        STAMP_TIMER_PT := UINT#0;
                        (* ! REGION TIMER[](STAMP_TIMER_IN, STAMP_TIMER_PT) => (STAMP_TIMER_ET, STAMP_TIMER_Q)
 *)                            IF STAMP_TIMER_IN THEN
                                STAMP_TIMER_Q := (STAMP_TIMER_ET = UINT#0);
                                IF (STAMP_TIMER_ET > UINT#0) THEN
                                    STAMP_TIMER_ET := (STAMP_TIMER_ET - UINT#1);
                                ELSE
                                    STAMP_TIMER_ET := UINT#0;
                                END_IF;
                            ELSE
                                STAMP_TIMER_Q := FALSE;
                                STAMP_TIMER_ET := STAMP_TIMER_PT;
                            END_IF;
                        (* ! END_REGION
 *)                        (* END OF ACTION CALL: STAMPSLIDERFORWARD_ACTIVE
 *)
                        IF STAMP_STAMPSLIDERMOVEDOUT THEN
                            STAMP_2_TRANSIT := TRUE;
                            STAMP_2STATE := STATES_STAMP#STEP2;
                        END_IF;

                    STATES_STAMP#STEP2:
                        STAMP_2_TRANSIT := FALSE;
                        IF (STAMP_CRANEONCONVEYOR AND NOT STAMP_STAMPSLIDERFILLED) THEN
                            STAMP_2_TRANSIT := TRUE;
                            STAMP_2STATE := STATES_STAMP#INTERSTEP;
                        END_IF;

                                    END_CASE;
                (* END OF: EDU.KIT.ITI.FORMAL.AUTOMATION.ST.TRANSLATIONSFCTOSTOLD_THEBIGSTATECASE
 *)
                (* RUNNING PIPELINE STEP: EDU.KIT.ITI.FORMAL.AUTOMATION.ST.SFCFLAGINTRODUCTION
 *)
            END_IF;
            (* END OF: EDU.KIT.ITI.FORMAL.AUTOMATION.ST.SFCFLAGINTRODUCTION
 *)
        (* ! END_REGION
 *)        IF (ACTUATOR_MAGAZINGREENLAMP AND ACTUATOR_STAMPGREENLAMP) THEN
            IF ((STAMP_STARTCOMMANDSTAMP AND CRANE_STARTCOMMANDCRANE) AND MAG_STARTCOMMANDMAGAZIN) THEN
                CRANE_STARTVAR := TRUE;
                MAG_STARTVAR := TRUE;
                STAMP_STARTVAR := TRUE;
            END_IF;
        END_IF;
        CRANE_SFCRESET := FALSE;
        MAG_SFCRESET := FALSE;
        STAMP_SFCRESET := FALSE;
    ELSIF (NOT SENSOR_STAMPEMERGENCYSTOP OR NOT SENSOR_MAGAZINEMERGENCYSTOP) THEN
        ACTUATOR_MAGAZINSLIDER := FALSE;
        ACTUATOR_CRANELOWER := FALSE;
        ACTUATOR_MAGAZINVACUUMON := FALSE;
        ACTUATOR_MAGAZINVACUUMOFF := TRUE;
        ACTUATOR_MAGAZINGREENLAMP := FALSE;
        ACTUATOR_CRANETURNCOUNTERCLOCKWISE := FALSE;
        ACTUATOR_CRANETURNCLOCKWISE := FALSE;
        ACTUATOR_STAMPSLIDERMOVEDOUT := TRUE;
        ACTUATOR_STAMPSLIDERMOVEDIN := FALSE;
        ACTUATOR_STAMPGREENLAMP := FALSE;
        ACTUATOR_STAMPPUSHER := FALSE;
        ACTUATOR_ANALOGCRANEPRESSURE := INT#0;
        CRANE_SFCRESET := TRUE;
        MAG_SFCRESET := TRUE;
        STAMP_SFCRESET := TRUE;
        CRANE_STARTVAR := FALSE;
        MAG_STARTVAR := FALSE;
        STAMP_STARTVAR := FALSE;
    END_IF;
END_PROGRAM

CONFIGURATION Config0
  RESOURCE Res0 ON PLC
    TASK TASK0(INTERVAL := T#50MS, PRIORITY := 0);
    PROGRAM INSTANCE0 WITH TASK0 : MAIN;
  END_RESOURCE
END_CONFIGURATION

(* ---- Scenario3v1_Final.xml.st0.st ---- *)
TYPE
    Stamp_states_t : (Green_Lamp , Init , Interstep , Interstep_2 , StampProcess , StampSliderBack , StampSliderForward , Stamp_Init_1 , Stamp_Init_2 , Stamp_Init_3 , Stamp_Init_4 , Start_Stamp , Step0 , Step1 , Step2);
    Magazin_states_t : (Green_Lamp , Init , Interstep , Magazin_Init , Magazin_Init_2 , Slider_Move_Back , Start_Magazin , Step0 , Step1 , convey);
    Crane_states_t : (Crane_Go_Up , Crane_Init , Crane_Init_2 , Crane_Lift_At_Stamp , Crane_Lift_Conveyor , Crane_Lift_Magazin , Crane_Lift_Magazin_Metallic , Crane_Lower , Crane_On_Conveyor , Crane_On_Conveyor_Metallic , Crane_On_Stamp_Metallic , Crane_Turn_Left_From_Stamp , Crane_Turn_Left_Metallic , Crane_Turn_Left_NOT_Metallic , Init , Interstep , Interstep_2 , Interstep_Check_Workpiece , Lower_Crane , Reset_interconnect , Start_Crane , Step0 , Step2 , Suck_At_Stamp , TimeDelay , Turn_Right , Wait_At_Stamp , pause , release , release_Workpiece);
END_TYPE

PROGRAM Main

VAR  Actuator_AnalogCranePressure : INT; END_VAR
VAR  Actuator_CraneLower : BOOL; END_VAR
VAR  Actuator_CraneTurnClockwise : BOOL; END_VAR
VAR  Actuator_CraneTurnCounterclockwise : BOOL; END_VAR
VAR  Actuator_MagazinGreenLamp : BOOL; END_VAR
VAR  Actuator_MagazinSlider : BOOL; END_VAR
VAR  Actuator_MagazinVacuumOff : BOOL; END_VAR
VAR  Actuator_MagazinVacuumOn : BOOL; END_VAR
VAR  Actuator_MagazinWhiteLamp : BOOL; END_VAR
VAR  Actuator_SomeActuator : BOOL; END_VAR
VAR  Actuator_StampGreenLamp : BOOL; END_VAR
VAR  Actuator_StampPusher : BOOL; END_VAR
VAR  Actuator_StampSliderMovedIn : BOOL; END_VAR
VAR  Actuator_StampSliderMovedOut : BOOL; END_VAR
VAR  Actuator_StampWhiteLamp : BOOL; END_VAR
VAR_INPUT  Crane_CraneDown : BOOL; END_VAR
VAR_OUTPUT  Crane_CraneLower : BOOL; END_VAR
VAR_INPUT  Crane_CraneOnConveyor : BOOL; END_VAR
VAR_INPUT  Crane_CraneOnMagazin : BOOL; END_VAR
VAR_INPUT  Crane_CranePositionStamp : BOOL; END_VAR
VAR_INPUT  Crane_CraneSucked : BOOL; END_VAR
VAR_OUTPUT  Crane_CraneTurnClockwise : BOOL; END_VAR
VAR_OUTPUT  Crane_CraneTurnCounterclockwise : BOOL; END_VAR
VAR_INPUT  Crane_CraneUp : BOOL; END_VAR
VAR  Crane_Duration1 : UINT := UINT#375; END_VAR
VAR_INPUT  Crane_MagazinCapacitiveSensor : BOOL; END_VAR
VAR_OUTPUT  Crane_MagazinVacuumOff : BOOL; END_VAR
VAR_OUTPUT  Crane_MagazinVacuumOn : BOOL; END_VAR
VAR  Crane_SFCInit : BOOL; END_VAR
VAR_INPUT  Crane_SFCReset : BOOL; END_VAR
VAR_INPUT  Crane_SliderMovedOut : BOOL; END_VAR
VAR_INPUT  Crane_SliderNotMovedOut : BOOL; END_VAR
VAR_INPUT  Crane_StampLowered : BOOL; END_VAR
VAR_INPUT  Crane_StampSliderFilled : BOOL; END_VAR
VAR_INPUT  Crane_StartButtonMagazin : BOOL; END_VAR
VAR_OUTPUT  Crane_StartCommandCrane : BOOL; END_VAR
VAR_INPUT  Crane_StartVar : BOOL; END_VAR
VAR_OUTPUT  Crane_TimeDelay_Timer_ET : USINT; END_VAR
VAR_INPUT  Crane_TimeDelay_Timer_IN : BOOL; END_VAR
VAR_INPUT  Crane_TimeDelay_Timer_PT : USINT; END_VAR
VAR_OUTPUT  Crane_TimeDelay_Timer_Q : BOOL; END_VAR
VAR  Crane_TimeDelay_Timer_Duration : UINT := UINT#12; END_VAR
VAR  Crane_TimeDelay_Timer_interconnect : BOOL; END_VAR
VAR_OUTPUT  Crane_Timer1_ET : USINT; END_VAR
VAR_INPUT  Crane_Timer1_IN : BOOL; END_VAR
VAR_INPUT  Crane_Timer1_PT : USINT; END_VAR
VAR_OUTPUT  Crane_Timer1_Q : BOOL; END_VAR
VAR_INPUT  Crane_WorkpieceReady : BOOL; END_VAR
VAR  Crane_2state : Crane_states_t; END_VAR
VAR  Crane_2transit : BOOL; END_VAR
VAR  Crane_actualtime1 : INT; END_VAR
VAR  Crane_interconnect : BOOL; END_VAR
VAR  Crane_interconnectCraneStartCommand : BOOL; END_VAR
VAR_INPUT  Mag_CraneDown : BOOL; END_VAR
VAR_OUTPUT  Mag_CraneLower : BOOL; END_VAR
VAR_INPUT  Mag_CraneOnConveyor : BOOL; END_VAR
VAR_INPUT  Mag_CraneOnMagazin : BOOL; END_VAR
VAR_INPUT  Mag_CraneSucked : BOOL; END_VAR
VAR_OUTPUT  Mag_CraneTurnClockwise : BOOL; END_VAR
VAR_OUTPUT  Mag_CraneTurnCounterclockwise : BOOL; END_VAR
VAR_INPUT  Mag_CraneUp : BOOL; END_VAR
VAR_OUTPUT  Mag_MagazinGreenLamp : BOOL; END_VAR
VAR_OUTPUT  Mag_MagazinSlider : BOOL; END_VAR
VAR_OUTPUT  Mag_MagazinVacuumOff : BOOL; END_VAR
VAR_OUTPUT  Mag_MagazinVacuumOn : BOOL; END_VAR
VAR_OUTPUT  Mag_MagazinWhiteLamp : BOOL; END_VAR
VAR  Mag_SFCInit : BOOL; END_VAR
VAR_INPUT  Mag_SFCReset : BOOL; END_VAR
VAR_INPUT  Mag_SliderMovedOut : BOOL; END_VAR
VAR_INPUT  Mag_SliderNotMovedOut : BOOL; END_VAR
VAR_INPUT  Mag_StartButtonMagazin : BOOL; END_VAR
VAR_OUTPUT  Mag_StartCommandMagazin : BOOL; END_VAR
VAR_INPUT  Mag_StartVar : BOOL; END_VAR
VAR_INPUT  Mag_WorkpieceReady : BOOL; END_VAR
VAR  Mag_2state : Magazin_states_t; END_VAR
VAR  Mag_2transit : BOOL; END_VAR
VAR  Mag_interconnectMagazinStartCommand : BOOL; END_VAR
VAR  Sensor_CraneDown : BOOL; END_VAR
VAR  Sensor_CraneOnConveyor : BOOL; END_VAR
VAR  Sensor_CraneOnMagazin : BOOL; END_VAR
VAR  Sensor_CranePosition : BOOL; END_VAR
VAR  Sensor_CranePositionStamp : BOOL; END_VAR
VAR  Sensor_CraneSucked : BOOL; END_VAR
VAR  Sensor_CraneUp : BOOL; END_VAR
VAR  Sensor_MagazinCapacitiveSensor : BOOL; END_VAR
VAR  Sensor_MagazinEmergencyStop : BOOL; END_VAR
VAR  Sensor_MagazinOpticalSensor : BOOL; END_VAR
VAR  Sensor_MagazinSwitchManuellAutomatic : BOOL; END_VAR
VAR  Sensor_SliderMovedOut : BOOL; END_VAR
VAR  Sensor_SliderNotMovedOut : BOOL; END_VAR
VAR  Sensor_StampEmergencyStop : BOOL; END_VAR
VAR  Sensor_StampLowered : BOOL; END_VAR
VAR  Sensor_StampSliderFilled : BOOL; END_VAR
VAR  Sensor_StampSliderSensorMovedIn : BOOL; END_VAR
VAR  Sensor_StampSliderSensorMovedOut : BOOL; END_VAR
VAR  Sensor_StampStartButton : BOOL; END_VAR
VAR  Sensor_StampSwitchManuellAutomatic : BOOL; END_VAR
VAR  Sensor_StampUp : BOOL; END_VAR
VAR  Sensor_StartButtonMagazin : BOOL; END_VAR
VAR  Sensor_WorkpieceReady : BOOL; END_VAR
VAR_INPUT  Stamp_CraneDown : BOOL; END_VAR
VAR_INPUT  Stamp_CraneOnConveyor : BOOL; END_VAR
VAR_INPUT  Stamp_CranePositionStamp : BOOL; END_VAR
VAR_INPUT  Stamp_CraneSucked : BOOL; END_VAR
VAR_INPUT  Stamp_CraneUp : BOOL; END_VAR
VAR  Stamp_Duration : UINT := UINT#125; END_VAR
VAR  Stamp_SFCInit : BOOL; END_VAR
VAR_INPUT  Stamp_SFCReset : BOOL; END_VAR
VAR_OUTPUT  Stamp_StampGreenLamp : BOOL; END_VAR
VAR_INPUT  Stamp_StampLowered : BOOL; END_VAR
VAR_OUTPUT  Stamp_StampPressure : BOOL; END_VAR
VAR_OUTPUT  Stamp_StampPusher : BOOL; END_VAR
VAR_INPUT  Stamp_StampSliderFilled : BOOL; END_VAR
VAR_OUTPUT  Stamp_StampSliderMovedIn : BOOL; END_VAR
VAR_OUTPUT  Stamp_StampSliderMovedOut : BOOL; END_VAR
VAR_INPUT  Stamp_StampSliderSensorMovedIn : BOOL; END_VAR
VAR_INPUT  Stamp_StampSliderSensorMovedOut : BOOL; END_VAR
VAR_INPUT  Stamp_StampStartButton : BOOL; END_VAR
VAR_INPUT  Stamp_StampUp : BOOL; END_VAR
VAR_OUTPUT  Stamp_StampWhiteLamp : BOOL; END_VAR
VAR_OUTPUT  Stamp_StartCommandStamp : BOOL; END_VAR
VAR_INPUT  Stamp_StartVar : BOOL; END_VAR
VAR_OUTPUT  Stamp_Timer_ET : USINT; END_VAR
VAR_INPUT  Stamp_Timer_IN : BOOL; END_VAR
VAR_INPUT  Stamp_Timer_PT : USINT; END_VAR
VAR_OUTPUT  Stamp_Timer_Q : BOOL; END_VAR
VAR  Stamp_2state : Stamp_states_t; END_VAR
VAR  Stamp_2transit : BOOL; END_VAR
VAR  Stamp_interconnect : BOOL; END_VAR
VAR  Stamp_interconnectStampStartCommand : BOOL; END_VAR
Mag_SliderNotMovedOut := Sensor_SliderNotMovedOut;
Mag_SliderMovedOut := Sensor_SliderMovedOut;
Mag_CraneOnMagazin := Sensor_CraneOnMagazin;
Mag_CraneDown := Sensor_CraneDown;
Mag_CraneUp := Sensor_CraneUp;
Mag_CraneOnConveyor := Sensor_CraneOnConveyor;
Mag_WorkpieceReady := Sensor_WorkpieceReady;
Mag_StartButtonMagazin := Sensor_StartButtonMagazin;
Actuator_MagazinSlider := Mag_MagazinSlider;
Actuator_MagazinGreenLamp := Mag_MagazinGreenLamp;
Crane_CraneUp := Sensor_CraneUp;
Crane_CraneOnConveyor := Sensor_CraneOnConveyor;
Crane_CraneDown := Sensor_CraneDown;
Crane_CraneSucked := Sensor_CraneSucked;
Crane_CraneOnMagazin := Sensor_CraneOnMagazin;
Crane_MagazinCapacitiveSensor := Sensor_MagazinCapacitiveSensor;
Crane_CranePositionStamp := Sensor_CranePositionStamp;
Crane_SliderMovedOut := Sensor_SliderMovedOut;
Crane_WorkpieceReady := Sensor_WorkpieceReady;
Crane_StampSliderFilled := Sensor_StampSliderFilled;
Crane_SliderMovedOut := Sensor_SliderMovedOut;
Crane_StartButtonMagazin := Sensor_StartButtonMagazin;
Actuator_CraneTurnCounterclockwise := Crane_CraneTurnCounterclockwise;
Actuator_CraneTurnClockwise := Crane_CraneTurnClockwise;
Actuator_CraneLower := Crane_CraneLower;
Actuator_MagazinVacuumOff := Crane_MagazinVacuumOff;
Actuator_MagazinVacuumOn := Crane_MagazinVacuumOn;
Stamp_StampSliderSensorMovedOut := Sensor_StampSliderSensorMovedOut;
Stamp_StampSliderSensorMovedIn := Sensor_StampSliderSensorMovedIn;
Stamp_StampSliderFilled := Sensor_StampSliderFilled;
Stamp_StampUp := Sensor_StampUp;
Stamp_StampLowered := Sensor_StampLowered;
Stamp_CraneDown := Sensor_CraneDown;
Stamp_CraneUp := Sensor_CraneUp;
Stamp_CraneSucked := Sensor_CraneSucked;
Stamp_CranePositionStamp := Sensor_CranePositionStamp;
Stamp_CraneOnConveyor := Sensor_CraneOnConveyor;
Stamp_StampStartButton := Sensor_StampStartButton;
Actuator_StampSliderMovedOut := Stamp_StampSliderMovedOut;
Actuator_StampSliderMovedIn := Stamp_StampSliderMovedIn;
Actuator_StampWhiteLamp := Stamp_StampWhiteLamp;
Actuator_StampPusher := Stamp_StampPusher;
Actuator_StampGreenLamp := Stamp_StampGreenLamp;
Actuator_AnalogCranePressure := INT#6000;
IF (Sensor_StampEmergencyStop AND Sensor_MagazinEmergencyStop) THEN
    CASE Mag_2state OF
        Magazin_states_t#Green_Lamp:

            Mag_2transit := FALSE;

            Mag_MagazinGreenLamp := TRUE;
            Mag_interconnectMagazinStartCommand := FALSE;

            IF TRUE THEN
                Mag_2transit := TRUE;
                Mag_2state := Magazin_states_t#Magazin_Init;
            END_IF;

        Magazin_states_t#Init:

            Mag_2transit := FALSE;

            IF TRUE THEN
                Mag_2transit := TRUE;
                Mag_2state := Magazin_states_t#Start_Magazin;
            END_IF;

        Magazin_states_t#Interstep:

            Mag_2transit := FALSE;

            Mag_StartCommandMagazin := TRUE;

            IF Mag_StartVar THEN
                Mag_2transit := TRUE;
                Mag_2state := Magazin_states_t#convey;
            END_IF;

        Magazin_states_t#Magazin_Init:

            Mag_2transit := FALSE;

            Mag_MagazinSlider := TRUE;

            IF TRUE THEN
                Mag_2transit := TRUE;
                Mag_2state := Magazin_states_t#Magazin_Init_2;
            END_IF;

        Magazin_states_t#Magazin_Init_2:

            Mag_2transit := FALSE;

            Mag_MagazinSlider := FALSE;

            IF TRUE THEN
                Mag_2transit := TRUE;
                Mag_2state := Magazin_states_t#Interstep;
            END_IF;

        Magazin_states_t#Slider_Move_Back:

            Mag_2transit := FALSE;

            IF ((Mag_SliderMovedOut = TRUE) AND (Mag_SliderNotMovedOut = FALSE)) THEN
                Mag_MagazinSlider := FALSE;
            END_IF;

            IF Mag_CraneUp THEN
                Mag_2transit := TRUE;
                Mag_2state := Magazin_states_t#Step1;
            END_IF;

        Magazin_states_t#Start_Magazin:

            Mag_2transit := FALSE;

            Mag_MagazinSlider := FALSE;
            Mag_MagazinGreenLamp := FALSE;
            Mag_StartVar := FALSE;
            Mag_StartCommandMagazin := FALSE;
            IF (Mag_StartButtonMagazin = TRUE) THEN
                Mag_interconnectMagazinStartCommand := TRUE;
            END_IF;

            IF Mag_interconnectMagazinStartCommand THEN
                Mag_2transit := TRUE;
                Mag_2state := Magazin_states_t#Green_Lamp;
            END_IF;

        Magazin_states_t#Step0:

            Mag_2transit := FALSE;

            IF Mag_CraneDown THEN
                Mag_2transit := TRUE;
                Mag_2state := Magazin_states_t#Slider_Move_Back;
            END_IF;

        Magazin_states_t#Step1:

            Mag_2transit := FALSE;

            IF Mag_CraneOnConveyor THEN
                Mag_2transit := TRUE;
                Mag_2state := Magazin_states_t#Interstep;
            END_IF;

        Magazin_states_t#convey:

            Mag_2transit := FALSE;

            IF Mag_SliderNotMovedOut THEN
                Mag_MagazinSlider := TRUE;
            END_IF;

            IF Mag_CraneOnMagazin THEN
                Mag_2transit := TRUE;
                Mag_2state := Magazin_states_t#Step0;
            END_IF;

            END_CASE;
    CASE Crane_2state OF
        Crane_states_t#Crane_Go_Up:

            Crane_2transit := FALSE;

            Crane_CraneLower := FALSE;

            IF Crane_CraneUp THEN
                Crane_2transit := TRUE;
                Crane_2state := Crane_states_t#pause;
            END_IF;

        Crane_states_t#Crane_Init:

            Crane_2transit := FALSE;

            Crane_CraneLower := TRUE;
            Crane_interconnectCraneStartCommand := FALSE;

            IF Crane_CraneDown THEN
                Crane_2transit := TRUE;
                Crane_2state := Crane_states_t#Crane_Init_2;
            END_IF;

        Crane_states_t#Crane_Init_2:

            Crane_2transit := FALSE;

            Crane_CraneLower := FALSE;

            IF Crane_CraneUp THEN
                Crane_2transit := TRUE;
                Crane_2state := Crane_states_t#Interstep;
            END_IF;

        Crane_states_t#Crane_Lift_At_Stamp:

            Crane_2transit := FALSE;

            Crane_CraneLower := FALSE;

            IF Crane_CraneUp THEN
                Crane_2transit := TRUE;
                Crane_2state := Crane_states_t#Crane_Turn_Left_From_Stamp;
            END_IF;

        Crane_states_t#Crane_Lift_Conveyor:

            Crane_2transit := FALSE;

            Crane_CraneLower := FALSE;

            IF TRUE THEN
                Crane_2transit := TRUE;
                Crane_2state := Crane_states_t#Interstep;
            END_IF;

        Crane_states_t#Crane_Lift_Magazin:

            Crane_2transit := FALSE;

            Crane_CraneLower := FALSE;

            IF Crane_CraneUp THEN
                Crane_2transit := TRUE;
                Crane_2state := Crane_states_t#Crane_Turn_Left_NOT_Metallic;
            END_IF;

        Crane_states_t#Crane_Lift_Magazin_Metallic:

            Crane_2transit := FALSE;

            Crane_CraneLower := FALSE;

            IF Crane_CraneUp THEN
                Crane_2transit := TRUE;
                Crane_2state := Crane_states_t#Crane_Turn_Left_Metallic;
            END_IF;

        Crane_states_t#Crane_Lower:

            Crane_2transit := FALSE;

            Crane_MagazinVacuumOn := TRUE;
            Crane_MagazinVacuumOff := FALSE;
            Crane_CraneLower := TRUE;

            IF Crane_CraneSucked THEN
                Crane_2transit := TRUE;
                Crane_2state := Crane_states_t#Step0;
            END_IF;

        Crane_states_t#Crane_On_Conveyor:

            Crane_2transit := FALSE;

            Crane_CraneTurnCounterclockwise := FALSE;
            Crane_CraneTurnClockwise := FALSE;
            Crane_CraneLower := TRUE;

            IF Crane_CraneDown THEN
                Crane_2transit := TRUE;
                Crane_2state := Crane_states_t#release;
            END_IF;

        Crane_states_t#Crane_On_Conveyor_Metallic:

            Crane_2transit := FALSE;

            Crane_CraneTurnCounterclockwise := FALSE;
            Crane_CraneTurnClockwise := FALSE;
            Crane_CraneLower := TRUE;

            IF Crane_CraneDown THEN
                Crane_2transit := TRUE;
                Crane_2state := Crane_states_t#release;
            END_IF;

        Crane_states_t#Crane_On_Stamp_Metallic:

            Crane_2transit := FALSE;

            Crane_CraneTurnCounterclockwise := FALSE;
            Crane_CraneTurnClockwise := FALSE;
            Crane_CraneLower := TRUE;

            IF Crane_CraneDown THEN
                Crane_2transit := TRUE;
                Crane_2state := Crane_states_t#release_Workpiece;
            END_IF;

        Crane_states_t#Crane_Turn_Left_From_Stamp:

            Crane_2transit := FALSE;

            Crane_CraneTurnClockwise := TRUE;
            Crane_CraneTurnCounterclockwise := FALSE;

            IF Crane_CraneOnConveyor THEN
                Crane_2transit := TRUE;
                Crane_2state := Crane_states_t#Crane_On_Conveyor_Metallic;
            END_IF;

        Crane_states_t#Crane_Turn_Left_Metallic:

            Crane_2transit := FALSE;

            Crane_CraneTurnCounterclockwise := TRUE;
            Crane_CraneTurnClockwise := FALSE;

            IF Crane_CranePositionStamp THEN
                Crane_2transit := TRUE;
                Crane_2state := Crane_states_t#Crane_On_Stamp_Metallic;
            END_IF;

        Crane_states_t#Crane_Turn_Left_NOT_Metallic:

            Crane_2transit := FALSE;

            Crane_CraneTurnCounterclockwise := TRUE;
            Crane_CraneTurnClockwise := FALSE;

            IF Crane_CraneOnConveyor THEN
                Crane_2transit := TRUE;
                Crane_2state := Crane_states_t#Crane_On_Conveyor;
            END_IF;

        Crane_states_t#Init:

            Crane_2transit := FALSE;

            IF TRUE THEN
                Crane_2transit := TRUE;
                Crane_2state := Crane_states_t#Start_Crane;
            END_IF;

        Crane_states_t#Interstep:

            Crane_2transit := FALSE;

            Crane_StartCommandCrane := TRUE;

            IF Crane_StartVar THEN
                Crane_2transit := TRUE;
                Crane_2state := Crane_states_t#Interstep_2;
            END_IF;

        Crane_states_t#Interstep_2:

            Crane_2transit := FALSE;

            IF Crane_SliderMovedOut THEN
                Crane_2transit := TRUE;
                Crane_2state := Crane_states_t#TimeDelay;
            END_IF;

        Crane_states_t#Interstep_Check_Workpiece:

            Crane_2transit := FALSE;

            Crane_CraneTurnClockwise := FALSE;
            Crane_CraneTurnCounterClockwise := FALSE;

            IF Crane_WorkpieceReady THEN
                Crane_2transit := TRUE;
                Crane_2state := Crane_states_t#Crane_Lower;
            ELSIF (NOT Crane_WorkpieceReady AND NOT Crane_StampSliderFilled) THEN
                Crane_2transit := TRUE;
                Crane_2state := Crane_states_t#Step2;
            ELSIF (NOT Crane_WorkpieceReady AND Crane_StampSliderFilled) THEN
                Crane_2transit := TRUE;
                Crane_2state := Crane_states_t#Wait_At_Stamp;
            END_IF;

        Crane_states_t#Lower_Crane:

            Crane_2transit := FALSE;

            Crane_CraneLower := TRUE;

            IF Crane_CraneDown THEN
                Crane_2transit := TRUE;
                Crane_2state := Crane_states_t#Suck_At_Stamp;
            END_IF;

        Crane_states_t#Reset_interconnect:

            Crane_2transit := FALSE;

            Crane_interconnect := FALSE;
            Crane_Timer1_IN := FALSE;
            Crane_Timer1_PT := USINT#0;
            IF Crane_Timer1_IN THEN
                Crane_Timer1_Q := (Crane_Timer1_ET = USINT#0);
                IF (Crane_Timer1_ET > USINT#0) THEN
                    Crane_Timer1_ET := (Crane_Timer1_ET - USINT#1);
                ELSE
                    Crane_Timer1_ET := USINT#0;
                END_IF;
            ELSE
                Crane_Timer1_Q := FALSE;
                Crane_Timer1_ET := Crane_Timer1_PT;
            END_IF;

            IF Crane_SliderMovedOut THEN
                Crane_2transit := TRUE;
                Crane_2state := Crane_states_t#Lower_Crane;
            END_IF;

        Crane_states_t#Start_Crane:

            Crane_2transit := FALSE;

            Crane_CraneLower := FALSE;
            Crane_MagazinVacuumOff := TRUE;
            Crane_MagazinVacuumOn := FALSE;
            Crane_CraneTurnCounterclockwise := FALSE;
            Crane_CraneTurnClockwise := FALSE;
            Crane_StartVar := FALSE;
            Crane_StartCommandCrane := FALSE;
            IF (Crane_StartButtonMagazin = TRUE) THEN
                Crane_interconnectCraneStartCommand := TRUE;
            END_IF;

            IF Crane_interconnectCraneStartCommand THEN
                Crane_2transit := TRUE;
                Crane_2state := Crane_states_t#Crane_Init;
            END_IF;

        Crane_states_t#Step0:

            Crane_2transit := FALSE;

            IF NOT Crane_MagazinCapacitiveSensor THEN
                Crane_2transit := TRUE;
                Crane_2state := Crane_states_t#Crane_Lift_Magazin;
            ELSIF Crane_MagazinCapacitiveSensor THEN
                Crane_2transit := TRUE;
                Crane_2state := Crane_states_t#Crane_Lift_Magazin_Metallic;
            END_IF;

        Crane_states_t#Step2:

            Crane_2transit := FALSE;

            IF TRUE THEN
                Crane_2transit := TRUE;
                Crane_2state := Crane_states_t#Start_Crane;
            END_IF;

        Crane_states_t#Suck_At_Stamp:

            Crane_2transit := FALSE;

            Crane_MagazinVacuumOn := TRUE;
            Crane_MagazinVacuumOff := FALSE;

            IF Crane_CraneSucked THEN
                Crane_2transit := TRUE;
                Crane_2state := Crane_states_t#Crane_Lift_At_Stamp;
            END_IF;

        Crane_states_t#TimeDelay:

            Crane_2transit := FALSE;

            Crane_TimeDelay_Timer_IN := TRUE;
            Crane_TimeDelay_Timer_PT := UINT_TO_USINT(Crane_TimeDelay_Timer_Duration);
            IF Crane_TimeDelay_Timer_IN THEN
                Crane_TimeDelay_Timer_Q := (Crane_TimeDelay_Timer_ET = USINT#0);
                IF (Crane_TimeDelay_Timer_ET > USINT#0) THEN
                    Crane_TimeDelay_Timer_ET := (Crane_TimeDelay_Timer_ET - USINT#1);
                ELSE
                    Crane_TimeDelay_Timer_ET := USINT#0;
                END_IF;
            ELSE
                Crane_TimeDelay_Timer_Q := FALSE;
                Crane_TimeDelay_Timer_ET := Crane_TimeDelay_Timer_PT;
            END_IF;
            Crane_TimeDelay_Timer_interconnect := Crane_TimeDelay_Timer_Q;

            IF Crane_TimeDelay_Timer_interconnect THEN
                Crane_2transit := TRUE;
                Crane_2state := Crane_states_t#Turn_Right;
            END_IF;

        Crane_states_t#Turn_Right:

            Crane_2transit := FALSE;

            Crane_CraneTurnClockwise := TRUE;
            Crane_CraneTurnCounterclockwise := FALSE;

            IF Crane_CraneOnMagazin THEN
                Crane_2transit := TRUE;
                Crane_2state := Crane_states_t#Interstep_Check_Workpiece;
            END_IF;

        Crane_states_t#Wait_At_Stamp:

            Crane_2transit := FALSE;

            IF TRUE THEN
                Crane_2transit := TRUE;
                Crane_2state := Crane_states_t#pause;
            END_IF;

        Crane_states_t#pause:

            Crane_2transit := FALSE;

            Crane_Timer1_IN := Crane_CraneUp;
            Crane_Timer1_PT := UINT_TO_USINT(Crane_Duration1);
            IF Crane_Timer1_IN THEN
                Crane_Timer1_Q := (Crane_Timer1_ET = USINT#0);
                IF (Crane_Timer1_ET > USINT#0) THEN
                    Crane_Timer1_ET := (Crane_Timer1_ET - USINT#1);
                ELSE
                    Crane_Timer1_ET := USINT#0;
                END_IF;
            ELSE
                Crane_Timer1_Q := FALSE;
                Crane_Timer1_ET := Crane_Timer1_PT;
            END_IF;
            Crane_interconnect := Crane_Timer1_Q;

            IF Crane_interconnect THEN
                Crane_2transit := TRUE;
                Crane_2state := Crane_states_t#Reset_interconnect;
            END_IF;

        Crane_states_t#release:

            Crane_2transit := FALSE;

            Crane_MagazinVacuumOff := TRUE;
            Crane_MagazinVacuumOn := FALSE;

            IF TRUE THEN
                Crane_2transit := TRUE;
                Crane_2state := Crane_states_t#Crane_Lift_Conveyor;
            END_IF;

        Crane_states_t#release_Workpiece:

            Crane_2transit := FALSE;

            Crane_MagazinVacuumOff := TRUE;
            Crane_MagazinVacuumOn := FALSE;

            IF TRUE THEN
                Crane_2transit := TRUE;
                Crane_2state := Crane_states_t#Crane_Go_Up;
            END_IF;

            END_CASE;
    CASE Stamp_2state OF
        Stamp_states_t#Green_Lamp:

            Stamp_2transit := FALSE;

            Stamp_StampGreenLamp := TRUE;
            Stamp_interconnectStampStartCommand := FALSE;

            IF TRUE THEN
                Stamp_2transit := TRUE;
                Stamp_2state := Stamp_states_t#Stamp_Init_1;
            END_IF;

        Stamp_states_t#Init:

            Stamp_2transit := FALSE;

            IF TRUE THEN
                Stamp_2transit := TRUE;
                Stamp_2state := Stamp_states_t#Start_Stamp;
            END_IF;

        Stamp_states_t#Interstep:

            Stamp_2transit := FALSE;

            Stamp_StartCommandStamp := TRUE;

            IF Stamp_StartVar THEN
                Stamp_2transit := TRUE;
                Stamp_2state := Stamp_states_t#Interstep_2;
            END_IF;

        Stamp_states_t#Interstep_2:

            Stamp_2transit := FALSE;

            IF Stamp_StampSliderFilled THEN
                Stamp_2transit := TRUE;
                Stamp_2state := Stamp_states_t#Step0;
            END_IF;

        Stamp_states_t#StampProcess:

            Stamp_2transit := FALSE;

            Stamp_StampSliderMovedIn := FALSE;
            Stamp_StampPusher := TRUE;

            IF Stamp_StampLowered THEN
                Stamp_2transit := TRUE;
                Stamp_2state := Stamp_states_t#Step1;
            END_IF;

        Stamp_states_t#StampSliderBack:

            Stamp_2transit := FALSE;

            Stamp_StampSliderMovedIn := TRUE;
            Stamp_StampSliderMovedOut := FALSE;

            IF Stamp_StampSliderSensorMovedIn THEN
                Stamp_2transit := TRUE;
                Stamp_2state := Stamp_states_t#StampProcess;
            END_IF;

        Stamp_states_t#StampSliderForward:

            Stamp_2transit := FALSE;

            Stamp_StampPusher := FALSE;
            Stamp_StampSliderMovedOut := TRUE;
            IF ((Stamp_StampLowered = FALSE) AND (Stamp_StampUp = TRUE)) THEN
                Stamp_interconnect := FALSE;
            END_IF;
            Stamp_Timer_IN := FALSE;
            Stamp_Timer_PT := USINT#0;
            IF Stamp_Timer_IN THEN
                Stamp_Timer_Q := (Stamp_Timer_ET = USINT#0);
                IF (Stamp_Timer_ET > USINT#0) THEN
                    Stamp_Timer_ET := (Stamp_Timer_ET - USINT#1);
                ELSE
                    Stamp_Timer_ET := USINT#0;
                END_IF;
            ELSE
                Stamp_Timer_Q := FALSE;
                Stamp_Timer_ET := Stamp_Timer_PT;
            END_IF;

            IF Stamp_StampSliderMovedOut THEN
                Stamp_2transit := TRUE;
                Stamp_2state := Stamp_states_t#Step2;
            END_IF;

        Stamp_states_t#Stamp_Init_1:

            Stamp_2transit := FALSE;

            Stamp_StampSliderMovedIn := TRUE;
            Stamp_StampSliderMovedOut := FALSE;

            IF Stamp_StampSliderSensorMovedIn THEN
                Stamp_2transit := TRUE;
                Stamp_2state := Stamp_states_t#Stamp_Init_2;
            END_IF;

        Stamp_states_t#Stamp_Init_2:

            Stamp_2transit := FALSE;

            Stamp_StampSliderMovedIn := FALSE;
            Stamp_StampSliderMovedOut := TRUE;

            IF Stamp_StampSliderSensorMovedOut THEN
                Stamp_2transit := TRUE;
                Stamp_2state := Stamp_states_t#Stamp_Init_3;
            END_IF;

        Stamp_states_t#Stamp_Init_3:

            Stamp_2transit := FALSE;

            Stamp_StampPusher := TRUE;

            IF Stamp_StampLowered THEN
                Stamp_2transit := TRUE;
                Stamp_2state := Stamp_states_t#Stamp_Init_4;
            END_IF;

        Stamp_states_t#Stamp_Init_4:

            Stamp_2transit := FALSE;

            Stamp_StampPusher := FALSE;

            IF Stamp_StampUp THEN
                Stamp_2transit := TRUE;
                Stamp_2state := Stamp_states_t#Interstep;
            END_IF;

        Stamp_states_t#Start_Stamp:

            Stamp_2transit := FALSE;

            Stamp_StampSliderMovedOut := FALSE;
            Stamp_StampSliderMovedIn := FALSE;
            Stamp_StampPusher := FALSE;
            Stamp_StampGreenLamp := FALSE;
            Stamp_StampPressure := FALSE;
            Stamp_StartCommandStamp := FALSE;
            IF (Stamp_StampStartButton = TRUE) THEN
                Stamp_interconnectStampStartCommand := TRUE;
            END_IF;

            IF Stamp_interconnectStampStartCommand THEN
                Stamp_2transit := TRUE;
                Stamp_2state := Stamp_states_t#Green_Lamp;
            END_IF;

        Stamp_states_t#Step0:

            Stamp_2transit := FALSE;

            IF Stamp_CraneUp THEN
                Stamp_2transit := TRUE;
                Stamp_2state := Stamp_states_t#StampSliderBack;
            END_IF;

        Stamp_states_t#Step1:

            Stamp_2transit := FALSE;

            Stamp_Timer_IN := Stamp_StampLowered;
            Stamp_Timer_PT := USINT#0;
            IF Stamp_Timer_IN THEN
                Stamp_Timer_Q := (Stamp_Timer_ET = USINT#0);
                IF (Stamp_Timer_ET > USINT#0) THEN
                    Stamp_Timer_ET := (Stamp_Timer_ET - USINT#1);
                ELSE
                    Stamp_Timer_ET := USINT#0;
                END_IF;
            ELSE
                Stamp_Timer_Q := FALSE;
                Stamp_Timer_ET := Stamp_Timer_PT;
            END_IF;
            Stamp_interconnect := Stamp_Timer_Q;

            IF Stamp_interconnect THEN
                Stamp_2transit := TRUE;
                Stamp_2state := Stamp_states_t#StampSliderForward;
            END_IF;

        Stamp_states_t#Step2:

            Stamp_2transit := FALSE;

            IF Stamp_CraneOnConveyor THEN
                Stamp_2transit := TRUE;
                Stamp_2state := Stamp_states_t#Interstep;
            END_IF;

            END_CASE;
    IF (Actuator_MagazinGreenLamp AND Actuator_StampGreenLamp) THEN
        IF ((Stamp_StartCommandStamp AND Crane_StartCommandCrane) AND Mag_StartCommandMagazin) THEN
            Crane_StartVar := TRUE;
            Mag_StartVar := TRUE;
            Stamp_StartVar := TRUE;
        END_IF;
    END_IF;
    Crane_SFCReset := FALSE;
    Mag_SFCReset := FALSE;
    Stamp_SFCReset := FALSE;
ELSIF (NOT Sensor_StampEmergencyStop OR NOT Sensor_MagazinEmergencyStop) THEN
    Actuator_MagazinSlider := FALSE;
    Actuator_CraneLower := FALSE;
    Actuator_MagazinVacuumOn := FALSE;
    Actuator_MagazinVacuumOff := TRUE;
    Actuator_MagazinGreenLamp := FALSE;
    Actuator_CraneTurnCounterclockwise := FALSE;
    Actuator_CraneTurnClockwise := FALSE;
    Actuator_StampSliderMovedOut := TRUE;
    Actuator_StampSliderMovedIn := FALSE;
    Actuator_StampGreenLamp := FALSE;
    Actuator_StampPusher := FALSE;
    Actuator_AnalogCranePressure := INT#0;
    Crane_SFCReset := TRUE;
    Mag_SFCReset := TRUE;
    Stamp_SFCReset := TRUE;
    Crane_StartVar := FALSE;
    Mag_StartVar := FALSE;
    Stamp_StartVar := FALSE;
END_IF;
END_PROGRAM
CONFIGURATION Config0
  RESOURCE Res0 ON PLC
    TASK task0(INTERVAL := T#50ms, PRIORITY := 0);
    PROGRAM instance0 WITH task0 : Main;
  END_RESOURCE
END_CONFIGURATION
